{attribute 'qualified_only'}
VAR_GLOBAL
	calc0: LREAL :=  10;
	calc1: LREAL :=  10;
	calc2: LREAL :=  10;
	calc3: LREAL :=  10;
	calc4: LREAL :=  10;
	calc5: LREAL :=  10;
	calc6: LREAL :=  10;
	calc7: LREAL :=  10;
	calc8: LREAL :=  10;
	calc9: LREAL :=  10;
	calc10: LREAL :=  10;
	calc11: LREAL :=  10;
	calc12: LREAL :=  10;
	calc13: LREAL :=  10;
	calc14: LREAL :=  10;
	calc15: LREAL :=  10;
	calc16: LREAL :=  10;
	calc17: LREAL :=  10;
	calc18: LREAL :=  10;
	calc19: LREAL :=  10;
	calc20: LREAL :=  10;
	calc21: LREAL :=  10;
	calc22: LREAL :=  10;
	calc23: LREAL :=  10;
	calc24: LREAL :=  10;
	calc25: LREAL :=  10;
	calc26: LREAL :=  10;
	calc27: LREAL :=  10;
	calc28: LREAL :=  10;
	calc29: LREAL :=  10;
	calc30: LREAL :=  10;
	calc31: LREAL :=  10;
	calc32: LREAL :=  10;
	calc33: LREAL :=  10;
	calc34: LREAL :=  10;
	calc35: LREAL :=  10;
	calc36: LREAL :=  10;
	calc37: LREAL :=  10;
	calc38: LREAL :=  10;
	calc39: LREAL :=  10;
	calc40: LREAL :=  10;
	calc41: LREAL :=  10;
	calc42: LREAL :=  10;
	calc43: LREAL :=  10;
	calc44: LREAL :=  10;
	calc45: LREAL :=  10;
	calc46: LREAL :=  10;
	calc47: LREAL :=  10;
	calc48: LREAL :=  10;
	calc49: LREAL :=  10;
	calc50: LREAL :=  10;
	calc51: LREAL :=  10;
	calc52: LREAL :=  10;
	calc53: LREAL :=  10;
	calc54: LREAL :=  10;
	calc55: LREAL :=  10;
	calc56: LREAL :=  10;
	calc57: LREAL :=  10;
	calc58: LREAL :=  10;
	calc59: LREAL :=  10;
	calc60: LREAL :=  10;
	calc61: LREAL :=  10;
	calc62: LREAL :=  10;
	calc63: LREAL :=  10;
	calc64: LREAL :=  10;
	calc65: LREAL :=  10;
	calc66: LREAL :=  10;
	calc67: LREAL :=  10;
	calc68: LREAL :=  10;
	calc69: LREAL :=  10;
	calc70: LREAL :=  10;
	calc71: LREAL :=  10;
	calc72: LREAL :=  10;
	calc73: LREAL :=  10;
	calc74: LREAL :=  10;
	calc75: LREAL :=  10;
	calc76: LREAL :=  10;
	calc77: LREAL :=  10;
	calc78: LREAL :=  10;
	calc79: LREAL :=  10;
	calc80: LREAL :=  10;
	calc81: LREAL :=  10;
	calc82: LREAL :=  10;
	calc83: LREAL :=  10;
	calc84: LREAL :=  10;
	calc85: LREAL :=  10;
	calc86: LREAL :=  10;
	calc87: LREAL :=  10;
	calc88: LREAL :=  10;
	calc89: LREAL :=  10;
	calc90: LREAL :=  10;
	calc91: LREAL :=  10;
	calc92: LREAL :=  10;
	calc93: LREAL :=  10;
	calc94: LREAL :=  10;
	calc95: LREAL :=  10;
	calc96: LREAL :=  10;
	calc97: LREAL :=  10;
	calc98: LREAL :=  10;
	calc99: LREAL :=  10;
	calc100: LREAL :=  10;
	calc101: LREAL :=  10;
	calc102: LREAL :=  10;
	calc103: LREAL :=  10;
	calc104: LREAL :=  10;
	calc105: LREAL :=  10;
	calc106: LREAL :=  10;
	calc107: LREAL :=  10;
	calc108: LREAL :=  10;
	calc109: LREAL :=  10;
	calc110: LREAL :=  10;
	calc111: LREAL :=  10;
	calc112: LREAL :=  10;
	calc113: LREAL :=  10;
	calc114: LREAL :=  10;
	calc115: LREAL :=  10;
	calc116: LREAL :=  10;
	calc117: LREAL :=  10;
	calc118: LREAL :=  10;
	calc119: LREAL :=  10;
	calc120: LREAL :=  10;
	calc121: LREAL :=  10;
	calc122: LREAL :=  10;
	calc123: LREAL :=  10;
	calc124: LREAL :=  10;
	calc125: LREAL :=  10;
	calc126: LREAL :=  10;
	calc127: LREAL :=  10;
	calc128: LREAL :=  10;
	calc129: LREAL :=  10;
	calc130: LREAL :=  10;
	calc131: LREAL :=  10;
	calc132: LREAL :=  10;
	calc133: LREAL :=  10;
	calc134: LREAL :=  10;
	calc135: LREAL :=  10;
	calc136: LREAL :=  10;
	calc137: LREAL :=  10;
	calc138: LREAL :=  10;
	calc139: LREAL :=  10;
	calc140: LREAL :=  10;
	calc141: LREAL :=  10;
	calc142: LREAL :=  10;
	calc143: LREAL :=  10;
	calc144: LREAL :=  10;
	calc145: LREAL :=  10;
	calc146: LREAL :=  10;
	calc147: LREAL :=  10;
	calc148: LREAL :=  10;
	calc149: LREAL :=  10;
	calc150: LREAL :=  10;
	calc151: LREAL :=  10;
	calc152: LREAL :=  10;
	calc153: LREAL :=  10;
	calc154: LREAL :=  10;
	calc155: LREAL :=  10;
	calc156: LREAL :=  10;
	calc157: LREAL :=  10;
	calc158: LREAL :=  10;
	calc159: LREAL :=  10;
	calc160: LREAL :=  10;
	calc161: LREAL :=  10;
	calc162: LREAL :=  10;
	calc163: LREAL :=  10;
	calc164: LREAL :=  10;
	calc165: LREAL :=  10;
	calc166: LREAL :=  10;
	calc167: LREAL :=  10;
	calc168: LREAL :=  10;
	calc169: LREAL :=  10;
	calc170: LREAL :=  10;
	calc171: LREAL :=  10;
	calc172: LREAL :=  10;
	calc173: LREAL :=  10;
	calc174: LREAL :=  10;
	calc175: LREAL :=  10;
	calc176: LREAL :=  10;
	calc177: LREAL :=  10;
	calc178: LREAL :=  10;
	calc179: LREAL :=  10;
	calc180: LREAL :=  10;
	calc181: LREAL :=  10;
	calc182: LREAL :=  10;
	calc183: LREAL :=  10;
	calc184: LREAL :=  10;
	calc185: LREAL :=  10;
	calc186: LREAL :=  10;
	calc187: LREAL :=  10;
	calc188: LREAL :=  10;
	calc189: LREAL :=  10;
	calc190: LREAL :=  10;
	calc191: LREAL :=  10;
	calc192: LREAL :=  10;
	calc193: LREAL :=  10;
	calc194: LREAL :=  10;
	calc195: LREAL :=  10;
	calc196: LREAL :=  10;
	calc197: LREAL :=  10;
	calc198: LREAL :=  10;
	calc199: LREAL :=  10;
	calc200: LREAL :=  10;
	calc201: LREAL :=  10;
	calc202: LREAL :=  10;
	calc203: LREAL :=  10;
	calc204: LREAL :=  10;
	calc205: LREAL :=  10;
	calc206: LREAL :=  10;
	calc207: LREAL :=  10;
	calc208: LREAL :=  10;
	calc209: LREAL :=  10;
	calc210: LREAL :=  10;
	calc211: LREAL :=  10;
	calc212: LREAL :=  10;
	calc213: LREAL :=  10;
	calc214: LREAL :=  10;
	calc215: LREAL :=  10;
	calc216: LREAL :=  10;
	calc217: LREAL :=  10;
	calc218: LREAL :=  10;
	calc219: LREAL :=  10;
	calc220: LREAL :=  10;
	calc221: LREAL :=  10;
	calc222: LREAL :=  10;
	calc223: LREAL :=  10;
	calc224: LREAL :=  10;
	calc225: LREAL :=  10;
	calc226: LREAL :=  10;
	calc227: LREAL :=  10;
	calc228: LREAL :=  10;
	calc229: LREAL :=  10;
	calc230: LREAL :=  10;
	calc231: LREAL :=  10;
	calc232: LREAL :=  10;
	calc233: LREAL :=  10;
	calc234: LREAL :=  10;
	calc235: LREAL :=  10;
	calc236: LREAL :=  10;
	calc237: LREAL :=  10;
	calc238: LREAL :=  10;
	calc239: LREAL :=  10;
	calc240: LREAL :=  10;
	calc241: LREAL :=  10;
	calc242: LREAL :=  10;
	calc243: LREAL :=  10;
	calc244: LREAL :=  10;
	calc245: LREAL :=  10;
	calc246: LREAL :=  10;
	calc247: LREAL :=  10;
	calc248: LREAL :=  10;
	calc249: LREAL :=  10;
	calc250: LREAL :=  10;
	calc251: LREAL :=  10;
	calc252: LREAL :=  10;
	calc253: LREAL :=  10;
	calc254: LREAL :=  10;
	calc255: LREAL :=  10;
	calc256: LREAL :=  10;
	calc257: LREAL :=  10;
	calc258: LREAL :=  10;
	calc259: LREAL :=  10;
	calc260: LREAL :=  10;
	calc261: LREAL :=  10;
	calc262: LREAL :=  10;
	calc263: LREAL :=  10;
	calc264: LREAL :=  10;
	calc265: LREAL :=  10;
	calc266: LREAL :=  10;
	calc267: LREAL :=  10;
	calc268: LREAL :=  10;
	calc269: LREAL :=  10;
	calc270: LREAL :=  10;
	calc271: LREAL :=  10;
	calc272: LREAL :=  10;
	calc273: LREAL :=  10;
	calc274: LREAL :=  10;
	calc275: LREAL :=  10;
	calc276: LREAL :=  10;
	calc277: LREAL :=  10;
	calc278: LREAL :=  10;
	calc279: LREAL :=  10;
	calc280: LREAL :=  10;
	calc281: LREAL :=  10;
	calc282: LREAL :=  10;
	calc283: LREAL :=  10;
	calc284: LREAL :=  10;
	calc285: LREAL :=  10;
	calc286: LREAL :=  10;
	calc287: LREAL :=  10;
	calc288: LREAL :=  10;
	calc289: LREAL :=  10;
	calc290: LREAL :=  10;
	calc291: LREAL :=  10;
	calc292: LREAL :=  10;
	calc293: LREAL :=  10;
	calc294: LREAL :=  10;
	calc295: LREAL :=  10;
	calc296: LREAL :=  10;
	calc297: LREAL :=  10;
	calc298: LREAL :=  10;
	calc299: LREAL :=  10;
	calc300: LREAL :=  10;
	calc301: LREAL :=  10;
	calc302: LREAL :=  10;
	calc303: LREAL :=  10;
	calc304: LREAL :=  10;
	calc305: LREAL :=  10;
	calc306: LREAL :=  10;
	calc307: LREAL :=  10;
	calc308: LREAL :=  10;
	calc309: LREAL :=  10;
	calc310: LREAL :=  10;
	calc311: LREAL :=  10;
	calc312: LREAL :=  10;
	calc313: LREAL :=  10;
	calc314: LREAL :=  10;
	calc315: LREAL :=  10;
	calc316: LREAL :=  10;
	calc317: LREAL :=  10;
	calc318: LREAL :=  10;
	calc319: LREAL :=  10;
	calc320: LREAL :=  10;
	calc321: LREAL :=  10;
	calc322: LREAL :=  10;
	calc323: LREAL :=  10;
	calc324: LREAL :=  10;
	calc325: LREAL :=  10;
	calc326: LREAL :=  10;
	calc327: LREAL :=  10;
	calc328: LREAL :=  10;
	calc329: LREAL :=  10;
	calc330: LREAL :=  10;
	calc331: LREAL :=  10;
	calc332: LREAL :=  10;
	calc333: LREAL :=  10;
	calc334: LREAL :=  10;
	calc335: LREAL :=  10;
	calc336: LREAL :=  10;
	calc337: LREAL :=  10;
	calc338: LREAL :=  10;
	calc339: LREAL :=  10;
	calc340: LREAL :=  10;
	calc341: LREAL :=  10;
	calc342: LREAL :=  10;
	calc343: LREAL :=  10;
	calc344: LREAL :=  10;
	calc345: LREAL :=  10;
	calc346: LREAL :=  10;
	calc347: LREAL :=  10;
	calc348: LREAL :=  10;
	calc349: LREAL :=  10;
	calc350: LREAL :=  10;
	calc351: LREAL :=  10;
	calc352: LREAL :=  10;
	calc353: LREAL :=  10;
	calc354: LREAL :=  10;
	calc355: LREAL :=  10;
	calc356: LREAL :=  10;
	calc357: LREAL :=  10;
	calc358: LREAL :=  10;
	calc359: LREAL :=  10;
	calc360: LREAL :=  10;
	calc361: LREAL :=  10;
	calc362: LREAL :=  10;
	calc363: LREAL :=  10;
	calc364: LREAL :=  10;
	calc365: LREAL :=  10;
	calc366: LREAL :=  10;
	calc367: LREAL :=  10;
	calc368: LREAL :=  10;
	calc369: LREAL :=  10;
	calc370: LREAL :=  10;
	calc371: LREAL :=  10;
	calc372: LREAL :=  10;
	calc373: LREAL :=  10;
	calc374: LREAL :=  10;
	calc375: LREAL :=  10;
	calc376: LREAL :=  10;
	calc377: LREAL :=  10;
	calc378: LREAL :=  10;
	calc379: LREAL :=  10;
	calc380: LREAL :=  10;
	calc381: LREAL :=  10;
	calc382: LREAL :=  10;
	calc383: LREAL :=  10;
	calc384: LREAL :=  10;
	calc385: LREAL :=  10;
	calc386: LREAL :=  10;
	calc387: LREAL :=  10;
	calc388: LREAL :=  10;
	calc389: LREAL :=  10;
	calc390: LREAL :=  10;
	calc391: LREAL :=  10;
	calc392: LREAL :=  10;
	calc393: LREAL :=  10;
	calc394: LREAL :=  10;
	calc395: LREAL :=  10;
	calc396: LREAL :=  10;
	calc397: LREAL :=  10;
	calc398: LREAL :=  10;
	calc399: LREAL :=  10;
	calc400: LREAL :=  10;
	calc401: LREAL :=  10;
	calc402: LREAL :=  10;
	calc403: LREAL :=  10;
	calc404: LREAL :=  10;
	calc405: LREAL :=  10;
	calc406: LREAL :=  10;
	calc407: LREAL :=  10;
	calc408: LREAL :=  10;
	calc409: LREAL :=  10;
	calc410: LREAL :=  10;
	calc411: LREAL :=  10;
	calc412: LREAL :=  10;
	calc413: LREAL :=  10;
	calc414: LREAL :=  10;
	calc415: LREAL :=  10;
	calc416: LREAL :=  10;
	calc417: LREAL :=  10;
	calc418: LREAL :=  10;
	calc419: LREAL :=  10;
	calc420: LREAL :=  10;
	calc421: LREAL :=  10;
	calc422: LREAL :=  10;
	calc423: LREAL :=  10;
	calc424: LREAL :=  10;
	calc425: LREAL :=  10;
	calc426: LREAL :=  10;
	calc427: LREAL :=  10;
	calc428: LREAL :=  10;
	calc429: LREAL :=  10;
	calc430: LREAL :=  10;
	calc431: LREAL :=  10;
	calc432: LREAL :=  10;
	calc433: LREAL :=  10;
	calc434: LREAL :=  10;
	calc435: LREAL :=  10;
	calc436: LREAL :=  10;
	calc437: LREAL :=  10;
	calc438: LREAL :=  10;
	calc439: LREAL :=  10;
	calc440: LREAL :=  10;
	calc441: LREAL :=  10;
	calc442: LREAL :=  10;
	calc443: LREAL :=  10;
	calc444: LREAL :=  10;
	calc445: LREAL :=  10;
	calc446: LREAL :=  10;
	calc447: LREAL :=  10;
	calc448: LREAL :=  10;
	calc449: LREAL :=  10;
	calc450: LREAL :=  10;
	calc451: LREAL :=  10;
	calc452: LREAL :=  10;
	calc453: LREAL :=  10;
	calc454: LREAL :=  10;
	calc455: LREAL :=  10;
	calc456: LREAL :=  10;
	calc457: LREAL :=  10;
	calc458: LREAL :=  10;
	calc459: LREAL :=  10;
	calc460: LREAL :=  10;
	calc461: LREAL :=  10;
	calc462: LREAL :=  10;
	calc463: LREAL :=  10;
	calc464: LREAL :=  10;
	calc465: LREAL :=  10;
	calc466: LREAL :=  10;
	calc467: LREAL :=  10;
	calc468: LREAL :=  10;
	calc469: LREAL :=  10;
	calc470: LREAL :=  10;
	calc471: LREAL :=  10;
	calc472: LREAL :=  10;
	calc473: LREAL :=  10;
	calc474: LREAL :=  10;
	calc475: LREAL :=  10;
	calc476: LREAL :=  10;
	calc477: LREAL :=  10;
	calc478: LREAL :=  10;
	calc479: LREAL :=  10;
	calc480: LREAL :=  10;
	calc481: LREAL :=  10;
	calc482: LREAL :=  10;
	calc483: LREAL :=  10;
	calc484: LREAL :=  10;
	calc485: LREAL :=  10;
	calc486: LREAL :=  10;
	calc487: LREAL :=  10;
	calc488: LREAL :=  10;
	calc489: LREAL :=  10;
	calc490: LREAL :=  10;
	calc491: LREAL :=  10;
	calc492: LREAL :=  10;
	calc493: LREAL :=  10;
	calc494: LREAL :=  10;
	calc495: LREAL :=  10;
	calc496: LREAL :=  10;
	calc497: LREAL :=  10;
	calc498: LREAL :=  10;
	calc499: LREAL :=  10;
	calc500: LREAL :=  10;
	calc501: LREAL :=  10;
	calc502: LREAL :=  10;
	calc503: LREAL :=  10;
	calc504: LREAL :=  10;
	calc505: LREAL :=  10;
	calc506: LREAL :=  10;
	calc507: LREAL :=  10;
	calc508: LREAL :=  10;
	calc509: LREAL :=  10;
	calc510: LREAL :=  10;
	calc511: LREAL :=  10;
	calc512: LREAL :=  10;
	calc513: LREAL :=  10;
	calc514: LREAL :=  10;
	calc515: LREAL :=  10;
	calc516: LREAL :=  10;
	calc517: LREAL :=  10;
	calc518: LREAL :=  10;
	calc519: LREAL :=  10;
	calc520: LREAL :=  10;
	calc521: LREAL :=  10;
	calc522: LREAL :=  10;
	calc523: LREAL :=  10;
	calc524: LREAL :=  10;
	calc525: LREAL :=  10;
	calc526: LREAL :=  10;
	calc527: LREAL :=  10;
	calc528: LREAL :=  10;
	calc529: LREAL :=  10;
	calc530: LREAL :=  10;
	calc531: LREAL :=  10;
	calc532: LREAL :=  10;
	calc533: LREAL :=  10;
	calc534: LREAL :=  10;
	calc535: LREAL :=  10;
	calc536: LREAL :=  10;
	calc537: LREAL :=  10;
	calc538: LREAL :=  10;
	calc539: LREAL :=  10;
	calc540: LREAL :=  10;
	calc541: LREAL :=  10;
	calc542: LREAL :=  10;
	calc543: LREAL :=  10;
	calc544: LREAL :=  10;
	calc545: LREAL :=  10;
	calc546: LREAL :=  10;
	calc547: LREAL :=  10;
	calc548: LREAL :=  10;
	calc549: LREAL :=  10;
	calc550: LREAL :=  10;
	calc551: LREAL :=  10;
	calc552: LREAL :=  10;
	calc553: LREAL :=  10;
	calc554: LREAL :=  10;
	calc555: LREAL :=  10;
	calc556: LREAL :=  10;
	calc557: LREAL :=  10;
	calc558: LREAL :=  10;
	calc559: LREAL :=  10;
	calc560: LREAL :=  10;
	calc561: LREAL :=  10;
	calc562: LREAL :=  10;
	calc563: LREAL :=  10;
	calc564: LREAL :=  10;
	calc565: LREAL :=  10;
	calc566: LREAL :=  10;
	calc567: LREAL :=  10;
	calc568: LREAL :=  10;
	calc569: LREAL :=  10;
	calc570: LREAL :=  10;
	calc571: LREAL :=  10;
	calc572: LREAL :=  10;
	calc573: LREAL :=  10;
	calc574: LREAL :=  10;
	calc575: LREAL :=  10;
	calc576: LREAL :=  10;
	calc577: LREAL :=  10;
	calc578: LREAL :=  10;
	calc579: LREAL :=  10;
	calc580: LREAL :=  10;
	calc581: LREAL :=  10;
	calc582: LREAL :=  10;
	calc583: LREAL :=  10;
	calc584: LREAL :=  10;
	calc585: LREAL :=  10;
	calc586: LREAL :=  10;
	calc587: LREAL :=  10;
	calc588: LREAL :=  10;
	calc589: LREAL :=  10;
	calc590: LREAL :=  10;
	calc591: LREAL :=  10;
	calc592: LREAL :=  10;
	calc593: LREAL :=  10;
	calc594: LREAL :=  10;
	calc595: LREAL :=  10;
	calc596: LREAL :=  10;
	calc597: LREAL :=  10;
	calc598: LREAL :=  10;
	calc599: LREAL :=  10;
	calc600: LREAL :=  10;
	calc601: LREAL :=  10;
	calc602: LREAL :=  10;
	calc603: LREAL :=  10;
	calc604: LREAL :=  10;
	calc605: LREAL :=  10;
	calc606: LREAL :=  10;
	calc607: LREAL :=  10;
	calc608: LREAL :=  10;
	calc609: LREAL :=  10;
	calc610: LREAL :=  10;
	calc611: LREAL :=  10;
	calc612: LREAL :=  10;
	calc613: LREAL :=  10;
	calc614: LREAL :=  10;
	calc615: LREAL :=  10;
	calc616: LREAL :=  10;
	calc617: LREAL :=  10;
	calc618: LREAL :=  10;
	calc619: LREAL :=  10;
	calc620: LREAL :=  10;
	calc621: LREAL :=  10;
	calc622: LREAL :=  10;
	calc623: LREAL :=  10;
	calc624: LREAL :=  10;
	calc625: LREAL :=  10;
	calc626: LREAL :=  10;
	calc627: LREAL :=  10;
	calc628: LREAL :=  10;
	calc629: LREAL :=  10;
	calc630: LREAL :=  10;
	calc631: LREAL :=  10;
	calc632: LREAL :=  10;
	calc633: LREAL :=  10;
	calc634: LREAL :=  10;
	calc635: LREAL :=  10;
	calc636: LREAL :=  10;
	calc637: LREAL :=  10;
	calc638: LREAL :=  10;
	calc639: LREAL :=  10;
	calc640: LREAL :=  10;
	calc641: LREAL :=  10;
	calc642: LREAL :=  10;
	calc643: LREAL :=  10;
	calc644: LREAL :=  10;
	calc645: LREAL :=  10;
	calc646: LREAL :=  10;
	calc647: LREAL :=  10;
	calc648: LREAL :=  10;
	calc649: LREAL :=  10;
	calc650: LREAL :=  10;
	calc651: LREAL :=  10;
	calc652: LREAL :=  10;
	calc653: LREAL :=  10;
	calc654: LREAL :=  10;
	calc655: LREAL :=  10;
	calc656: LREAL :=  10;
	calc657: LREAL :=  10;
	calc658: LREAL :=  10;
	calc659: LREAL :=  10;
	calc660: LREAL :=  10;
	calc661: LREAL :=  10;
	calc662: LREAL :=  10;
	calc663: LREAL :=  10;
	calc664: LREAL :=  10;
	calc665: LREAL :=  10;
	calc666: LREAL :=  10;
	calc667: LREAL :=  10;
	calc668: LREAL :=  10;
	calc669: LREAL :=  10;
	calc670: LREAL :=  10;
	calc671: LREAL :=  10;
	calc672: LREAL :=  10;
	calc673: LREAL :=  10;
	calc674: LREAL :=  10;
	calc675: LREAL :=  10;
	calc676: LREAL :=  10;
	calc677: LREAL :=  10;
	calc678: LREAL :=  10;
	calc679: LREAL :=  10;
	calc680: LREAL :=  10;
	calc681: LREAL :=  10;
	calc682: LREAL :=  10;
	calc683: LREAL :=  10;
	calc684: LREAL :=  10;
	calc685: LREAL :=  10;
	calc686: LREAL :=  10;
	calc687: LREAL :=  10;
	calc688: LREAL :=  10;
	calc689: LREAL :=  10;
	calc690: LREAL :=  10;
	calc691: LREAL :=  10;
	calc692: LREAL :=  10;
	calc693: LREAL :=  10;
	calc694: LREAL :=  10;
	calc695: LREAL :=  10;
	calc696: LREAL :=  10;
	calc697: LREAL :=  10;
	calc698: LREAL :=  10;
	calc699: LREAL :=  10;
	calc700: LREAL :=  10;
	calc701: LREAL :=  10;
	calc702: LREAL :=  10;
	calc703: LREAL :=  10;
	calc704: LREAL :=  10;
	calc705: LREAL :=  10;
	calc706: LREAL :=  10;
	calc707: LREAL :=  10;
	calc708: LREAL :=  10;
	calc709: LREAL :=  10;
	calc710: LREAL :=  10;
	calc711: LREAL :=  10;
	calc712: LREAL :=  10;
	calc713: LREAL :=  10;
	calc714: LREAL :=  10;
	calc715: LREAL :=  10;
	calc716: LREAL :=  10;
	calc717: LREAL :=  10;
	calc718: LREAL :=  10;
	calc719: LREAL :=  10;
	calc720: LREAL :=  10;
	calc721: LREAL :=  10;
	calc722: LREAL :=  10;
	calc723: LREAL :=  10;
	calc724: LREAL :=  10;
	calc725: LREAL :=  10;
	calc726: LREAL :=  10;
	calc727: LREAL :=  10;
	calc728: LREAL :=  10;
	calc729: LREAL :=  10;
	calc730: LREAL :=  10;
	calc731: LREAL :=  10;
	calc732: LREAL :=  10;
	calc733: LREAL :=  10;
	calc734: LREAL :=  10;
	calc735: LREAL :=  10;
	calc736: LREAL :=  10;
	calc737: LREAL :=  10;
	calc738: LREAL :=  10;
	calc739: LREAL :=  10;
	calc740: LREAL :=  10;
	calc741: LREAL :=  10;
	calc742: LREAL :=  10;
	calc743: LREAL :=  10;
	calc744: LREAL :=  10;
	calc745: LREAL :=  10;
	calc746: LREAL :=  10;
	calc747: LREAL :=  10;
	calc748: LREAL :=  10;
	calc749: LREAL :=  10;
	calc750: LREAL :=  10;
	calc751: LREAL :=  10;
	calc752: LREAL :=  10;
	calc753: LREAL :=  10;
	calc754: LREAL :=  10;
	calc755: LREAL :=  10;
	calc756: LREAL :=  10;
	calc757: LREAL :=  10;
	calc758: LREAL :=  10;
	calc759: LREAL :=  10;
	calc760: LREAL :=  10;
	calc761: LREAL :=  10;
	calc762: LREAL :=  10;
	calc763: LREAL :=  10;
	calc764: LREAL :=  10;
	calc765: LREAL :=  10;
	calc766: LREAL :=  10;
	calc767: LREAL :=  10;
	calc768: LREAL :=  10;
	calc769: LREAL :=  10;
	calc770: LREAL :=  10;
	calc771: LREAL :=  10;
	calc772: LREAL :=  10;
	calc773: LREAL :=  10;
	calc774: LREAL :=  10;
	calc775: LREAL :=  10;
	calc776: LREAL :=  10;
	calc777: LREAL :=  10;
	calc778: LREAL :=  10;
	calc779: LREAL :=  10;
	calc780: LREAL :=  10;
	calc781: LREAL :=  10;
	calc782: LREAL :=  10;
	calc783: LREAL :=  10;
	calc784: LREAL :=  10;
	calc785: LREAL :=  10;
	calc786: LREAL :=  10;
	calc787: LREAL :=  10;
	calc788: LREAL :=  10;
	calc789: LREAL :=  10;
	calc790: LREAL :=  10;
	calc791: LREAL :=  10;
	calc792: LREAL :=  10;
	calc793: LREAL :=  10;
	calc794: LREAL :=  10;
	calc795: LREAL :=  10;
	calc796: LREAL :=  10;
	calc797: LREAL :=  10;
	calc798: LREAL :=  10;
	calc799: LREAL :=  10;
	calc800: LREAL :=  10;
	calc801: LREAL :=  10;
	calc802: LREAL :=  10;
	calc803: LREAL :=  10;
	calc804: LREAL :=  10;
	calc805: LREAL :=  10;
	calc806: LREAL :=  10;
	calc807: LREAL :=  10;
	calc808: LREAL :=  10;
	calc809: LREAL :=  10;
	calc810: LREAL :=  10;
	calc811: LREAL :=  10;
	calc812: LREAL :=  10;
	calc813: LREAL :=  10;
	calc814: LREAL :=  10;
	calc815: LREAL :=  10;
	calc816: LREAL :=  10;
	calc817: LREAL :=  10;
	calc818: LREAL :=  10;
	calc819: LREAL :=  10;
	calc820: LREAL :=  10;
	calc821: LREAL :=  10;
	calc822: LREAL :=  10;
	calc823: LREAL :=  10;
	calc824: LREAL :=  10;
	calc825: LREAL :=  10;
	calc826: LREAL :=  10;
	calc827: LREAL :=  10;
	calc828: LREAL :=  10;
	calc829: LREAL :=  10;
	calc830: LREAL :=  10;
	calc831: LREAL :=  10;
	calc832: LREAL :=  10;
	calc833: LREAL :=  10;
	calc834: LREAL :=  10;
	calc835: LREAL :=  10;
	calc836: LREAL :=  10;
	calc837: LREAL :=  10;
	calc838: LREAL :=  10;
	calc839: LREAL :=  10;
	calc840: LREAL :=  10;
	calc841: LREAL :=  10;
	calc842: LREAL :=  10;
	calc843: LREAL :=  10;
	calc844: LREAL :=  10;
	calc845: LREAL :=  10;
	calc846: LREAL :=  10;
	calc847: LREAL :=  10;
	calc848: LREAL :=  10;
	calc849: LREAL :=  10;
	calc850: LREAL :=  10;
	calc851: LREAL :=  10;
	calc852: LREAL :=  10;
	calc853: LREAL :=  10;
	calc854: LREAL :=  10;
	calc855: LREAL :=  10;
	calc856: LREAL :=  10;
	calc857: LREAL :=  10;
	calc858: LREAL :=  10;
	calc859: LREAL :=  10;
	calc860: LREAL :=  10;
	calc861: LREAL :=  10;
	calc862: LREAL :=  10;
	calc863: LREAL :=  10;
	calc864: LREAL :=  10;
	calc865: LREAL :=  10;
	calc866: LREAL :=  10;
	calc867: LREAL :=  10;
	calc868: LREAL :=  10;
	calc869: LREAL :=  10;
	calc870: LREAL :=  10;
	calc871: LREAL :=  10;
	calc872: LREAL :=  10;
	calc873: LREAL :=  10;
	calc874: LREAL :=  10;
	calc875: LREAL :=  10;
	calc876: LREAL :=  10;
	calc877: LREAL :=  10;
	calc878: LREAL :=  10;
	calc879: LREAL :=  10;
	calc880: LREAL :=  10;
	calc881: LREAL :=  10;
	calc882: LREAL :=  10;
	calc883: LREAL :=  10;
	calc884: LREAL :=  10;
	calc885: LREAL :=  10;
	calc886: LREAL :=  10;
	calc887: LREAL :=  10;
	calc888: LREAL :=  10;
	calc889: LREAL :=  10;
	calc890: LREAL :=  10;
	calc891: LREAL :=  10;
	calc892: LREAL :=  10;
	calc893: LREAL :=  10;
	calc894: LREAL :=  10;
	calc895: LREAL :=  10;
	calc896: LREAL :=  10;
	calc897: LREAL :=  10;
	calc898: LREAL :=  10;
	calc899: LREAL :=  10;
	calc900: LREAL :=  10;
	calc901: LREAL :=  10;
	calc902: LREAL :=  10;
	calc903: LREAL :=  10;
	calc904: LREAL :=  10;
	calc905: LREAL :=  10;
	calc906: LREAL :=  10;
	calc907: LREAL :=  10;
	calc908: LREAL :=  10;
	calc909: LREAL :=  10;
	calc910: LREAL :=  10;
	calc911: LREAL :=  10;
	calc912: LREAL :=  10;
	calc913: LREAL :=  10;
	calc914: LREAL :=  10;
	calc915: LREAL :=  10;
	calc916: LREAL :=  10;
	calc917: LREAL :=  10;
	calc918: LREAL :=  10;
	calc919: LREAL :=  10;
	calc920: LREAL :=  10;
	calc921: LREAL :=  10;
	calc922: LREAL :=  10;
	calc923: LREAL :=  10;
	calc924: LREAL :=  10;
	calc925: LREAL :=  10;
	calc926: LREAL :=  10;
	calc927: LREAL :=  10;
	calc928: LREAL :=  10;
	calc929: LREAL :=  10;
	calc930: LREAL :=  10;
	calc931: LREAL :=  10;
	calc932: LREAL :=  10;
	calc933: LREAL :=  10;
	calc934: LREAL :=  10;
	calc935: LREAL :=  10;
	calc936: LREAL :=  10;
	calc937: LREAL :=  10;
	calc938: LREAL :=  10;
	calc939: LREAL :=  10;
	calc940: LREAL :=  10;
	calc941: LREAL :=  10;
	calc942: LREAL :=  10;
	calc943: LREAL :=  10;
	calc944: LREAL :=  10;
	calc945: LREAL :=  10;
	calc946: LREAL :=  10;
	calc947: LREAL :=  10;
	calc948: LREAL :=  10;
	calc949: LREAL :=  10;
	calc950: LREAL :=  10;
	calc951: LREAL :=  10;
	calc952: LREAL :=  10;
	calc953: LREAL :=  10;
	calc954: LREAL :=  10;
	calc955: LREAL :=  10;
	calc956: LREAL :=  10;
	calc957: LREAL :=  10;
	calc958: LREAL :=  10;
	calc959: LREAL :=  10;
	calc960: LREAL :=  10;
	calc961: LREAL :=  10;
	calc962: LREAL :=  10;
	calc963: LREAL :=  10;
	calc964: LREAL :=  10;
	calc965: LREAL :=  10;
	calc966: LREAL :=  10;
	calc967: LREAL :=  10;
	calc968: LREAL :=  10;
	calc969: LREAL :=  10;
	calc970: LREAL :=  10;
	calc971: LREAL :=  10;
	calc972: LREAL :=  10;
	calc973: LREAL :=  10;
	calc974: LREAL :=  10;
	calc975: LREAL :=  10;
	calc976: LREAL :=  10;
	calc977: LREAL :=  10;
	calc978: LREAL :=  10;
	calc979: LREAL :=  10;
	calc980: LREAL :=  10;
	calc981: LREAL :=  10;
	calc982: LREAL :=  10;
	calc983: LREAL :=  10;
	calc984: LREAL :=  10;
	calc985: LREAL :=  10;
	calc986: LREAL :=  10;
	calc987: LREAL :=  10;
	calc988: LREAL :=  10;
	calc989: LREAL :=  10;
	calc990: LREAL :=  10;
	calc991: LREAL :=  10;
	calc992: LREAL :=  10;
	calc993: LREAL :=  10;
	calc994: LREAL :=  10;
	calc995: LREAL :=  10;
	calc996: LREAL :=  10;
	calc997: LREAL :=  10;
	calc998: LREAL :=  10;
	calc999: LREAL :=  10;
	calc1000: LREAL :=  10;
	calc1001: LREAL :=  10;
	calc1002: LREAL :=  10;
	calc1003: LREAL :=  10;
	calc1004: LREAL :=  10;
	calc1005: LREAL :=  10;
	calc1006: LREAL :=  10;
	calc1007: LREAL :=  10;
	calc1008: LREAL :=  10;
	calc1009: LREAL :=  10;
	calc1010: LREAL :=  10;
	calc1011: LREAL :=  10;
	calc1012: LREAL :=  10;
	calc1013: LREAL :=  10;
	calc1014: LREAL :=  10;
	calc1015: LREAL :=  10;
	calc1016: LREAL :=  10;
	calc1017: LREAL :=  10;
	calc1018: LREAL :=  10;
	calc1019: LREAL :=  10;
	calc1020: LREAL :=  10;
	calc1021: LREAL :=  10;
	calc1022: LREAL :=  10;
	calc1023: LREAL :=  10;
	calc1024: LREAL :=  10;
	calc1025: LREAL :=  10;
	calc1026: LREAL :=  10;
	calc1027: LREAL :=  10;
	calc1028: LREAL :=  10;
	calc1029: LREAL :=  10;
	calc1030: LREAL :=  10;
	calc1031: LREAL :=  10;
	calc1032: LREAL :=  10;
	calc1033: LREAL :=  10;
	calc1034: LREAL :=  10;
	calc1035: LREAL :=  10;
	calc1036: LREAL :=  10;
	calc1037: LREAL :=  10;
	calc1038: LREAL :=  10;
	calc1039: LREAL :=  10;
	calc1040: LREAL :=  10;
	calc1041: LREAL :=  10;
	calc1042: LREAL :=  10;
	calc1043: LREAL :=  10;
	calc1044: LREAL :=  10;
	calc1045: LREAL :=  10;
	calc1046: LREAL :=  10;
	calc1047: LREAL :=  10;
	calc1048: LREAL :=  10;
	calc1049: LREAL :=  10;
	calc1050: LREAL :=  10;
	calc1051: LREAL :=  10;
	calc1052: LREAL :=  10;
	calc1053: LREAL :=  10;
	calc1054: LREAL :=  10;
	calc1055: LREAL :=  10;
	calc1056: LREAL :=  10;
	calc1057: LREAL :=  10;
	calc1058: LREAL :=  10;
	calc1059: LREAL :=  10;
	calc1060: LREAL :=  10;
	calc1061: LREAL :=  10;
	calc1062: LREAL :=  10;
	calc1063: LREAL :=  10;
	calc1064: LREAL :=  10;
	calc1065: LREAL :=  10;
	calc1066: LREAL :=  10;
	calc1067: LREAL :=  10;
	calc1068: LREAL :=  10;
	calc1069: LREAL :=  10;
	calc1070: LREAL :=  10;
	calc1071: LREAL :=  10;
	calc1072: LREAL :=  10;
	calc1073: LREAL :=  10;
	calc1074: LREAL :=  10;
	calc1075: LREAL :=  10;
	calc1076: LREAL :=  10;
	calc1077: LREAL :=  10;
	calc1078: LREAL :=  10;
	calc1079: LREAL :=  10;
	calc1080: LREAL :=  10;
	calc1081: LREAL :=  10;
	calc1082: LREAL :=  10;
	calc1083: LREAL :=  10;
	calc1084: LREAL :=  10;
	calc1085: LREAL :=  10;
	calc1086: LREAL :=  10;
	calc1087: LREAL :=  10;
	calc1088: LREAL :=  10;
	calc1089: LREAL :=  10;
	calc1090: LREAL :=  10;
	calc1091: LREAL :=  10;
	calc1092: LREAL :=  10;
	calc1093: LREAL :=  10;
	calc1094: LREAL :=  10;
	calc1095: LREAL :=  10;
	calc1096: LREAL :=  10;
	calc1097: LREAL :=  10;
	calc1098: LREAL :=  10;
	calc1099: LREAL :=  10;
	calc1100: LREAL :=  10;
	calc1101: LREAL :=  10;
	calc1102: LREAL :=  10;
	calc1103: LREAL :=  10;
	calc1104: LREAL :=  10;
	calc1105: LREAL :=  10;
	calc1106: LREAL :=  10;
	calc1107: LREAL :=  10;
	calc1108: LREAL :=  10;
	calc1109: LREAL :=  10;
	calc1110: LREAL :=  10;
	calc1111: LREAL :=  10;
	calc1112: LREAL :=  10;
	calc1113: LREAL :=  10;
	calc1114: LREAL :=  10;
	calc1115: LREAL :=  10;
	calc1116: LREAL :=  10;
	calc1117: LREAL :=  10;
	calc1118: LREAL :=  10;
	calc1119: LREAL :=  10;
	calc1120: LREAL :=  10;
	calc1121: LREAL :=  10;
	calc1122: LREAL :=  10;
	calc1123: LREAL :=  10;
	calc1124: LREAL :=  10;
	calc1125: LREAL :=  10;
	calc1126: LREAL :=  10;
	calc1127: LREAL :=  10;
	calc1128: LREAL :=  10;
	calc1129: LREAL :=  10;
	calc1130: LREAL :=  10;
	calc1131: LREAL :=  10;
	calc1132: LREAL :=  10;
	calc1133: LREAL :=  10;
	calc1134: LREAL :=  10;
	calc1135: LREAL :=  10;
	calc1136: LREAL :=  10;
	calc1137: LREAL :=  10;
	calc1138: LREAL :=  10;
	calc1139: LREAL :=  10;
	calc1140: LREAL :=  10;
	calc1141: LREAL :=  10;
	calc1142: LREAL :=  10;
	calc1143: LREAL :=  10;
	calc1144: LREAL :=  10;
	calc1145: LREAL :=  10;
	calc1146: LREAL :=  10;
	calc1147: LREAL :=  10;
	calc1148: LREAL :=  10;
	calc1149: LREAL :=  10;
	calc1150: LREAL :=  10;
	calc1151: LREAL :=  10;
	calc1152: LREAL :=  10;
	calc1153: LREAL :=  10;
	calc1154: LREAL :=  10;
	calc1155: LREAL :=  10;
	calc1156: LREAL :=  10;
	calc1157: LREAL :=  10;
	calc1158: LREAL :=  10;
	calc1159: LREAL :=  10;
	calc1160: LREAL :=  10;
	calc1161: LREAL :=  10;
	calc1162: LREAL :=  10;
	calc1163: LREAL :=  10;
	calc1164: LREAL :=  10;
	calc1165: LREAL :=  10;
	calc1166: LREAL :=  10;
	calc1167: LREAL :=  10;
	calc1168: LREAL :=  10;
	calc1169: LREAL :=  10;
	calc1170: LREAL :=  10;
	calc1171: LREAL :=  10;
	calc1172: LREAL :=  10;
	calc1173: LREAL :=  10;
	calc1174: LREAL :=  10;
	calc1175: LREAL :=  10;
	calc1176: LREAL :=  10;
	calc1177: LREAL :=  10;
	calc1178: LREAL :=  10;
	calc1179: LREAL :=  10;
	calc1180: LREAL :=  10;
	calc1181: LREAL :=  10;
	calc1182: LREAL :=  10;
	calc1183: LREAL :=  10;
	calc1184: LREAL :=  10;
	calc1185: LREAL :=  10;
	calc1186: LREAL :=  10;
	calc1187: LREAL :=  10;
	calc1188: LREAL :=  10;
	calc1189: LREAL :=  10;
	calc1190: LREAL :=  10;
	calc1191: LREAL :=  10;
	calc1192: LREAL :=  10;
	calc1193: LREAL :=  10;
	calc1194: LREAL :=  10;
	calc1195: LREAL :=  10;
	calc1196: LREAL :=  10;
	calc1197: LREAL :=  10;
	calc1198: LREAL :=  10;
	calc1199: LREAL :=  10;
	calc1200: LREAL :=  10;
	calc1201: LREAL :=  10;
	calc1202: LREAL :=  10;
	calc1203: LREAL :=  10;
	calc1204: LREAL :=  10;
	calc1205: LREAL :=  10;
	calc1206: LREAL :=  10;
	calc1207: LREAL :=  10;
	calc1208: LREAL :=  10;
	calc1209: LREAL :=  10;
	calc1210: LREAL :=  10;
	calc1211: LREAL :=  10;
	calc1212: LREAL :=  10;
	calc1213: LREAL :=  10;
	calc1214: LREAL :=  10;
	calc1215: LREAL :=  10;
	calc1216: LREAL :=  10;
	calc1217: LREAL :=  10;
	calc1218: LREAL :=  10;
	calc1219: LREAL :=  10;
	calc1220: LREAL :=  10;
	calc1221: LREAL :=  10;
	calc1222: LREAL :=  10;
	calc1223: LREAL :=  10;
	calc1224: LREAL :=  10;
	calc1225: LREAL :=  10;
	calc1226: LREAL :=  10;
	calc1227: LREAL :=  10;
	calc1228: LREAL :=  10;
	calc1229: LREAL :=  10;
	calc1230: LREAL :=  10;
	calc1231: LREAL :=  10;
	calc1232: LREAL :=  10;
	calc1233: LREAL :=  10;
	calc1234: LREAL :=  10;
	calc1235: LREAL :=  10;
	calc1236: LREAL :=  10;
	calc1237: LREAL :=  10;
	calc1238: LREAL :=  10;
	calc1239: LREAL :=  10;
	calc1240: LREAL :=  10;
	calc1241: LREAL :=  10;
	calc1242: LREAL :=  10;
	calc1243: LREAL :=  10;
	calc1244: LREAL :=  10;
	calc1245: LREAL :=  10;
	calc1246: LREAL :=  10;
	calc1247: LREAL :=  10;
	calc1248: LREAL :=  10;
	calc1249: LREAL :=  10;
	calc1250: LREAL :=  10;
	calc1251: LREAL :=  10;
	calc1252: LREAL :=  10;
	calc1253: LREAL :=  10;
	calc1254: LREAL :=  10;
	calc1255: LREAL :=  10;
	calc1256: LREAL :=  10;
	calc1257: LREAL :=  10;
	calc1258: LREAL :=  10;
	calc1259: LREAL :=  10;
	calc1260: LREAL :=  10;
	calc1261: LREAL :=  10;
	calc1262: LREAL :=  10;
	calc1263: LREAL :=  10;
	calc1264: LREAL :=  10;
	calc1265: LREAL :=  10;
	calc1266: LREAL :=  10;
	calc1267: LREAL :=  10;
	calc1268: LREAL :=  10;
	calc1269: LREAL :=  10;
	calc1270: LREAL :=  10;
	calc1271: LREAL :=  10;
	calc1272: LREAL :=  10;
	calc1273: LREAL :=  10;
	calc1274: LREAL :=  10;
	calc1275: LREAL :=  10;
	calc1276: LREAL :=  10;
	calc1277: LREAL :=  10;
	calc1278: LREAL :=  10;
	calc1279: LREAL :=  10;
	calc1280: LREAL :=  10;
	calc1281: LREAL :=  10;
	calc1282: LREAL :=  10;
	calc1283: LREAL :=  10;
	calc1284: LREAL :=  10;
	calc1285: LREAL :=  10;
	calc1286: LREAL :=  10;
	calc1287: LREAL :=  10;
	calc1288: LREAL :=  10;
	calc1289: LREAL :=  10;
	calc1290: LREAL :=  10;
	calc1291: LREAL :=  10;
	calc1292: LREAL :=  10;
	calc1293: LREAL :=  10;
	calc1294: LREAL :=  10;
	calc1295: LREAL :=  10;
	calc1296: LREAL :=  10;
	calc1297: LREAL :=  10;
	calc1298: LREAL :=  10;
	calc1299: LREAL :=  10;
	calc1300: LREAL :=  10;
	calc1301: LREAL :=  10;
	calc1302: LREAL :=  10;
	calc1303: LREAL :=  10;
	calc1304: LREAL :=  10;
	calc1305: LREAL :=  10;
	calc1306: LREAL :=  10;
	calc1307: LREAL :=  10;
	calc1308: LREAL :=  10;
	calc1309: LREAL :=  10;
	calc1310: LREAL :=  10;
	calc1311: LREAL :=  10;
	calc1312: LREAL :=  10;
	calc1313: LREAL :=  10;
	calc1314: LREAL :=  10;
	calc1315: LREAL :=  10;
	calc1316: LREAL :=  10;
	calc1317: LREAL :=  10;
	calc1318: LREAL :=  10;
	calc1319: LREAL :=  10;
	calc1320: LREAL :=  10;
	calc1321: LREAL :=  10;
	calc1322: LREAL :=  10;
	calc1323: LREAL :=  10;
	calc1324: LREAL :=  10;
	calc1325: LREAL :=  10;
	calc1326: LREAL :=  10;
	calc1327: LREAL :=  10;
	calc1328: LREAL :=  10;
	calc1329: LREAL :=  10;
	calc1330: LREAL :=  10;
	calc1331: LREAL :=  10;
	calc1332: LREAL :=  10;
	calc1333: LREAL :=  10;
	calc1334: LREAL :=  10;
	calc1335: LREAL :=  10;
	calc1336: LREAL :=  10;
	calc1337: LREAL :=  10;
	calc1338: LREAL :=  10;
	calc1339: LREAL :=  10;
	calc1340: LREAL :=  10;
	calc1341: LREAL :=  10;
	calc1342: LREAL :=  10;
	calc1343: LREAL :=  10;
	calc1344: LREAL :=  10;
	calc1345: LREAL :=  10;
	calc1346: LREAL :=  10;
	calc1347: LREAL :=  10;
	calc1348: LREAL :=  10;
	calc1349: LREAL :=  10;
	calc1350: LREAL :=  10;
	calc1351: LREAL :=  10;
	calc1352: LREAL :=  10;
	calc1353: LREAL :=  10;
	calc1354: LREAL :=  10;
	calc1355: LREAL :=  10;
	calc1356: LREAL :=  10;
	calc1357: LREAL :=  10;
	calc1358: LREAL :=  10;
	calc1359: LREAL :=  10;
	calc1360: LREAL :=  10;
	calc1361: LREAL :=  10;
	calc1362: LREAL :=  10;
	calc1363: LREAL :=  10;
	calc1364: LREAL :=  10;
	calc1365: LREAL :=  10;
	calc1366: LREAL :=  10;
	calc1367: LREAL :=  10;
	calc1368: LREAL :=  10;
	calc1369: LREAL :=  10;
	calc1370: LREAL :=  10;
	calc1371: LREAL :=  10;
	calc1372: LREAL :=  10;
	calc1373: LREAL :=  10;
	calc1374: LREAL :=  10;
	calc1375: LREAL :=  10;
	calc1376: LREAL :=  10;
	calc1377: LREAL :=  10;
	calc1378: LREAL :=  10;
	calc1379: LREAL :=  10;
	calc1380: LREAL :=  10;
	calc1381: LREAL :=  10;
	calc1382: LREAL :=  10;
	calc1383: LREAL :=  10;
	calc1384: LREAL :=  10;
	calc1385: LREAL :=  10;
	calc1386: LREAL :=  10;
	calc1387: LREAL :=  10;
	calc1388: LREAL :=  10;
	calc1389: LREAL :=  10;
	calc1390: LREAL :=  10;
	calc1391: LREAL :=  10;
	calc1392: LREAL :=  10;
	calc1393: LREAL :=  10;
	calc1394: LREAL :=  10;
	calc1395: LREAL :=  10;
	calc1396: LREAL :=  10;
	calc1397: LREAL :=  10;
	calc1398: LREAL :=  10;
	calc1399: LREAL :=  10;
	calc1400: LREAL :=  10;
	calc1401: LREAL :=  10;
	calc1402: LREAL :=  10;
	calc1403: LREAL :=  10;
	calc1404: LREAL :=  10;
	calc1405: LREAL :=  10;
	calc1406: LREAL :=  10;
	calc1407: LREAL :=  10;
	calc1408: LREAL :=  10;
	calc1409: LREAL :=  10;
	calc1410: LREAL :=  10;
	calc1411: LREAL :=  10;
	calc1412: LREAL :=  10;
	calc1413: LREAL :=  10;
	calc1414: LREAL :=  10;
	calc1415: LREAL :=  10;
	calc1416: LREAL :=  10;
	calc1417: LREAL :=  10;
	calc1418: LREAL :=  10;
	calc1419: LREAL :=  10;
	calc1420: LREAL :=  10;
	calc1421: LREAL :=  10;
	calc1422: LREAL :=  10;
	calc1423: LREAL :=  10;
	calc1424: LREAL :=  10;
	calc1425: LREAL :=  10;
	calc1426: LREAL :=  10;
	calc1427: LREAL :=  10;
	calc1428: LREAL :=  10;
	calc1429: LREAL :=  10;
	calc1430: LREAL :=  10;
	calc1431: LREAL :=  10;
	calc1432: LREAL :=  10;
	calc1433: LREAL :=  10;
	calc1434: LREAL :=  10;
	calc1435: LREAL :=  10;
	calc1436: LREAL :=  10;
	calc1437: LREAL :=  10;
	calc1438: LREAL :=  10;
	calc1439: LREAL :=  10;
	calc1440: LREAL :=  10;
	calc1441: LREAL :=  10;
	calc1442: LREAL :=  10;
	calc1443: LREAL :=  10;
	calc1444: LREAL :=  10;
	calc1445: LREAL :=  10;
	calc1446: LREAL :=  10;
	calc1447: LREAL :=  10;
	calc1448: LREAL :=  10;
	calc1449: LREAL :=  10;
	calc1450: LREAL :=  10;
	calc1451: LREAL :=  10;
	calc1452: LREAL :=  10;
	calc1453: LREAL :=  10;
	calc1454: LREAL :=  10;
	calc1455: LREAL :=  10;
	calc1456: LREAL :=  10;
	calc1457: LREAL :=  10;
	calc1458: LREAL :=  10;
	calc1459: LREAL :=  10;
	calc1460: LREAL :=  10;
	calc1461: LREAL :=  10;
	calc1462: LREAL :=  10;
	calc1463: LREAL :=  10;
	calc1464: LREAL :=  10;
	calc1465: LREAL :=  10;
	calc1466: LREAL :=  10;
	calc1467: LREAL :=  10;
	calc1468: LREAL :=  10;
	calc1469: LREAL :=  10;
	calc1470: LREAL :=  10;
	calc1471: LREAL :=  10;
	calc1472: LREAL :=  10;
	calc1473: LREAL :=  10;
	calc1474: LREAL :=  10;
	calc1475: LREAL :=  10;
	calc1476: LREAL :=  10;
	calc1477: LREAL :=  10;
	calc1478: LREAL :=  10;
	calc1479: LREAL :=  10;
	calc1480: LREAL :=  10;
	calc1481: LREAL :=  10;
	calc1482: LREAL :=  10;
	calc1483: LREAL :=  10;
	calc1484: LREAL :=  10;
	calc1485: LREAL :=  10;
	calc1486: LREAL :=  10;
	calc1487: LREAL :=  10;
	calc1488: LREAL :=  10;
	calc1489: LREAL :=  10;
	calc1490: LREAL :=  10;
	calc1491: LREAL :=  10;
	calc1492: LREAL :=  10;
	calc1493: LREAL :=  10;
	calc1494: LREAL :=  10;
	calc1495: LREAL :=  10;
	calc1496: LREAL :=  10;
	calc1497: LREAL :=  10;
	calc1498: LREAL :=  10;
	calc1499: LREAL :=  10;
	calc1500: LREAL :=  10;
	calc1501: LREAL :=  10;
	calc1502: LREAL :=  10;
	calc1503: LREAL :=  10;
	calc1504: LREAL :=  10;
	calc1505: LREAL :=  10;
	calc1506: LREAL :=  10;
	calc1507: LREAL :=  10;
	calc1508: LREAL :=  10;
	calc1509: LREAL :=  10;
	calc1510: LREAL :=  10;
	calc1511: LREAL :=  10;
	calc1512: LREAL :=  10;
	calc1513: LREAL :=  10;
	calc1514: LREAL :=  10;
	calc1515: LREAL :=  10;
	calc1516: LREAL :=  10;
	calc1517: LREAL :=  10;
	calc1518: LREAL :=  10;
	calc1519: LREAL :=  10;
	calc1520: LREAL :=  10;
	calc1521: LREAL :=  10;
	calc1522: LREAL :=  10;
	calc1523: LREAL :=  10;
	calc1524: LREAL :=  10;
	calc1525: LREAL :=  10;
	calc1526: LREAL :=  10;
	calc1527: LREAL :=  10;
	calc1528: LREAL :=  10;
	calc1529: LREAL :=  10;
	calc1530: LREAL :=  10;
	calc1531: LREAL :=  10;
	calc1532: LREAL :=  10;
	calc1533: LREAL :=  10;
	calc1534: LREAL :=  10;
	calc1535: LREAL :=  10;
	calc1536: LREAL :=  10;
	calc1537: LREAL :=  10;
	calc1538: LREAL :=  10;
	calc1539: LREAL :=  10;
	calc1540: LREAL :=  10;
	calc1541: LREAL :=  10;
	calc1542: LREAL :=  10;
	calc1543: LREAL :=  10;
	calc1544: LREAL :=  10;
	calc1545: LREAL :=  10;
	calc1546: LREAL :=  10;
	calc1547: LREAL :=  10;
	calc1548: LREAL :=  10;
	calc1549: LREAL :=  10;
	calc1550: LREAL :=  10;
	calc1551: LREAL :=  10;
	calc1552: LREAL :=  10;
	calc1553: LREAL :=  10;
	calc1554: LREAL :=  10;
	calc1555: LREAL :=  10;
	calc1556: LREAL :=  10;
	calc1557: LREAL :=  10;
	calc1558: LREAL :=  10;
	calc1559: LREAL :=  10;
	calc1560: LREAL :=  10;
	calc1561: LREAL :=  10;
	calc1562: LREAL :=  10;
	calc1563: LREAL :=  10;
	calc1564: LREAL :=  10;
	calc1565: LREAL :=  10;
	calc1566: LREAL :=  10;
	calc1567: LREAL :=  10;
	calc1568: LREAL :=  10;
	calc1569: LREAL :=  10;
	calc1570: LREAL :=  10;
	calc1571: LREAL :=  10;
	calc1572: LREAL :=  10;
	calc1573: LREAL :=  10;
	calc1574: LREAL :=  10;
	calc1575: LREAL :=  10;
	calc1576: LREAL :=  10;
	calc1577: LREAL :=  10;
	calc1578: LREAL :=  10;
	calc1579: LREAL :=  10;
	calc1580: LREAL :=  10;
	calc1581: LREAL :=  10;
	calc1582: LREAL :=  10;
	calc1583: LREAL :=  10;
	calc1584: LREAL :=  10;
	calc1585: LREAL :=  10;
	calc1586: LREAL :=  10;
	calc1587: LREAL :=  10;
	calc1588: LREAL :=  10;
	calc1589: LREAL :=  10;
	calc1590: LREAL :=  10;
	calc1591: LREAL :=  10;
	calc1592: LREAL :=  10;
	calc1593: LREAL :=  10;
	calc1594: LREAL :=  10;
	calc1595: LREAL :=  10;
	calc1596: LREAL :=  10;
	calc1597: LREAL :=  10;
	calc1598: LREAL :=  10;
	calc1599: LREAL :=  10;
	calc1600: LREAL :=  10;
	calc1601: LREAL :=  10;
	calc1602: LREAL :=  10;
	calc1603: LREAL :=  10;
	calc1604: LREAL :=  10;
	calc1605: LREAL :=  10;
	calc1606: LREAL :=  10;
	calc1607: LREAL :=  10;
	calc1608: LREAL :=  10;
	calc1609: LREAL :=  10;
	calc1610: LREAL :=  10;
	calc1611: LREAL :=  10;
	calc1612: LREAL :=  10;
	calc1613: LREAL :=  10;
	calc1614: LREAL :=  10;
	calc1615: LREAL :=  10;
	calc1616: LREAL :=  10;
	calc1617: LREAL :=  10;
	calc1618: LREAL :=  10;
	calc1619: LREAL :=  10;
	calc1620: LREAL :=  10;
	calc1621: LREAL :=  10;
	calc1622: LREAL :=  10;
	calc1623: LREAL :=  10;
	calc1624: LREAL :=  10;
	calc1625: LREAL :=  10;
	calc1626: LREAL :=  10;
	calc1627: LREAL :=  10;
	calc1628: LREAL :=  10;
	calc1629: LREAL :=  10;
	calc1630: LREAL :=  10;
	calc1631: LREAL :=  10;
	calc1632: LREAL :=  10;
	calc1633: LREAL :=  10;
	calc1634: LREAL :=  10;
	calc1635: LREAL :=  10;
	calc1636: LREAL :=  10;
	calc1637: LREAL :=  10;
	calc1638: LREAL :=  10;
	calc1639: LREAL :=  10;
	calc1640: LREAL :=  10;
	calc1641: LREAL :=  10;
	calc1642: LREAL :=  10;
	calc1643: LREAL :=  10;
	calc1644: LREAL :=  10;
	calc1645: LREAL :=  10;
	calc1646: LREAL :=  10;
	calc1647: LREAL :=  10;
	calc1648: LREAL :=  10;
	calc1649: LREAL :=  10;
	calc1650: LREAL :=  10;
	calc1651: LREAL :=  10;
	calc1652: LREAL :=  10;
	calc1653: LREAL :=  10;
	calc1654: LREAL :=  10;
	calc1655: LREAL :=  10;
	calc1656: LREAL :=  10;
	calc1657: LREAL :=  10;
	calc1658: LREAL :=  10;
	calc1659: LREAL :=  10;
	calc1660: LREAL :=  10;
	calc1661: LREAL :=  10;
	calc1662: LREAL :=  10;
	calc1663: LREAL :=  10;
	calc1664: LREAL :=  10;
	calc1665: LREAL :=  10;
	calc1666: LREAL :=  10;
	calc1667: LREAL :=  10;
	calc1668: LREAL :=  10;
	calc1669: LREAL :=  10;
	calc1670: LREAL :=  10;
	calc1671: LREAL :=  10;
	calc1672: LREAL :=  10;
	calc1673: LREAL :=  10;
	calc1674: LREAL :=  10;
	calc1675: LREAL :=  10;
	calc1676: LREAL :=  10;
	calc1677: LREAL :=  10;
	calc1678: LREAL :=  10;
	calc1679: LREAL :=  10;
	calc1680: LREAL :=  10;
	calc1681: LREAL :=  10;
	calc1682: LREAL :=  10;
	calc1683: LREAL :=  10;
	calc1684: LREAL :=  10;
	calc1685: LREAL :=  10;
	calc1686: LREAL :=  10;
	calc1687: LREAL :=  10;
	calc1688: LREAL :=  10;
	calc1689: LREAL :=  10;
	calc1690: LREAL :=  10;
	calc1691: LREAL :=  10;
	calc1692: LREAL :=  10;
	calc1693: LREAL :=  10;
	calc1694: LREAL :=  10;
	calc1695: LREAL :=  10;
	calc1696: LREAL :=  10;
	calc1697: LREAL :=  10;
	calc1698: LREAL :=  10;
	calc1699: LREAL :=  10;
	calc1700: LREAL :=  10;
	calc1701: LREAL :=  10;
	calc1702: LREAL :=  10;
	calc1703: LREAL :=  10;
	calc1704: LREAL :=  10;
	calc1705: LREAL :=  10;
	calc1706: LREAL :=  10;
	calc1707: LREAL :=  10;
	calc1708: LREAL :=  10;
	calc1709: LREAL :=  10;
	calc1710: LREAL :=  10;
	calc1711: LREAL :=  10;
	calc1712: LREAL :=  10;
	calc1713: LREAL :=  10;
	calc1714: LREAL :=  10;
	calc1715: LREAL :=  10;
	calc1716: LREAL :=  10;
	calc1717: LREAL :=  10;
	calc1718: LREAL :=  10;
	calc1719: LREAL :=  10;
	calc1720: LREAL :=  10;
	calc1721: LREAL :=  10;
	calc1722: LREAL :=  10;
	calc1723: LREAL :=  10;
	calc1724: LREAL :=  10;
	calc1725: LREAL :=  10;
	calc1726: LREAL :=  10;
	calc1727: LREAL :=  10;
	calc1728: LREAL :=  10;
	calc1729: LREAL :=  10;
	calc1730: LREAL :=  10;
	calc1731: LREAL :=  10;
	calc1732: LREAL :=  10;
	calc1733: LREAL :=  10;
	calc1734: LREAL :=  10;
	calc1735: LREAL :=  10;
	calc1736: LREAL :=  10;
	calc1737: LREAL :=  10;
	calc1738: LREAL :=  10;
	calc1739: LREAL :=  10;
	calc1740: LREAL :=  10;
	calc1741: LREAL :=  10;
	calc1742: LREAL :=  10;
	calc1743: LREAL :=  10;
	calc1744: LREAL :=  10;
	calc1745: LREAL :=  10;
	calc1746: LREAL :=  10;
	calc1747: LREAL :=  10;
	calc1748: LREAL :=  10;
	calc1749: LREAL :=  10;
	calc1750: LREAL :=  10;
	calc1751: LREAL :=  10;
	calc1752: LREAL :=  10;
	calc1753: LREAL :=  10;
	calc1754: LREAL :=  10;
	calc1755: LREAL :=  10;
	calc1756: LREAL :=  10;
	calc1757: LREAL :=  10;
	calc1758: LREAL :=  10;
	calc1759: LREAL :=  10;
	calc1760: LREAL :=  10;
	calc1761: LREAL :=  10;
	calc1762: LREAL :=  10;
	calc1763: LREAL :=  10;
	calc1764: LREAL :=  10;
	calc1765: LREAL :=  10;
	calc1766: LREAL :=  10;
	calc1767: LREAL :=  10;
	calc1768: LREAL :=  10;
	calc1769: LREAL :=  10;
	calc1770: LREAL :=  10;
	calc1771: LREAL :=  10;
	calc1772: LREAL :=  10;
	calc1773: LREAL :=  10;
	calc1774: LREAL :=  10;
	calc1775: LREAL :=  10;
	calc1776: LREAL :=  10;
	calc1777: LREAL :=  10;
	calc1778: LREAL :=  10;
	calc1779: LREAL :=  10;
	calc1780: LREAL :=  10;
	calc1781: LREAL :=  10;
	calc1782: LREAL :=  10;
	calc1783: LREAL :=  10;
	calc1784: LREAL :=  10;
	calc1785: LREAL :=  10;
	calc1786: LREAL :=  10;
	calc1787: LREAL :=  10;
	calc1788: LREAL :=  10;
	calc1789: LREAL :=  10;
	calc1790: LREAL :=  10;
	calc1791: LREAL :=  10;
	calc1792: LREAL :=  10;
	calc1793: LREAL :=  10;
	calc1794: LREAL :=  10;
	calc1795: LREAL :=  10;
	calc1796: LREAL :=  10;
	calc1797: LREAL :=  10;
	calc1798: LREAL :=  10;
	calc1799: LREAL :=  10;
	calc1800: LREAL :=  10;
	calc1801: LREAL :=  10;
	calc1802: LREAL :=  10;
	calc1803: LREAL :=  10;
	calc1804: LREAL :=  10;
	calc1805: LREAL :=  10;
	calc1806: LREAL :=  10;
	calc1807: LREAL :=  10;
	calc1808: LREAL :=  10;
	calc1809: LREAL :=  10;
	calc1810: LREAL :=  10;
	calc1811: LREAL :=  10;
	calc1812: LREAL :=  10;
	calc1813: LREAL :=  10;
	calc1814: LREAL :=  10;
	calc1815: LREAL :=  10;
	calc1816: LREAL :=  10;
	calc1817: LREAL :=  10;
	calc1818: LREAL :=  10;
	calc1819: LREAL :=  10;
	calc1820: LREAL :=  10;
	calc1821: LREAL :=  10;
	calc1822: LREAL :=  10;
	calc1823: LREAL :=  10;
	calc1824: LREAL :=  10;
	calc1825: LREAL :=  10;
	calc1826: LREAL :=  10;
	calc1827: LREAL :=  10;
	calc1828: LREAL :=  10;
	calc1829: LREAL :=  10;
	calc1830: LREAL :=  10;
	calc1831: LREAL :=  10;
	calc1832: LREAL :=  10;
	calc1833: LREAL :=  10;
	calc1834: LREAL :=  10;
	calc1835: LREAL :=  10;
	calc1836: LREAL :=  10;
	calc1837: LREAL :=  10;
	calc1838: LREAL :=  10;
	calc1839: LREAL :=  10;
	calc1840: LREAL :=  10;
	calc1841: LREAL :=  10;
	calc1842: LREAL :=  10;
	calc1843: LREAL :=  10;
	calc1844: LREAL :=  10;
	calc1845: LREAL :=  10;
	calc1846: LREAL :=  10;
	calc1847: LREAL :=  10;
	calc1848: LREAL :=  10;
	calc1849: LREAL :=  10;
	calc1850: LREAL :=  10;
	calc1851: LREAL :=  10;
	calc1852: LREAL :=  10;
	calc1853: LREAL :=  10;
	calc1854: LREAL :=  10;
	calc1855: LREAL :=  10;
	calc1856: LREAL :=  10;
	calc1857: LREAL :=  10;
	calc1858: LREAL :=  10;
	calc1859: LREAL :=  10;
	calc1860: LREAL :=  10;
	calc1861: LREAL :=  10;
	calc1862: LREAL :=  10;
	calc1863: LREAL :=  10;
	calc1864: LREAL :=  10;
	calc1865: LREAL :=  10;
	calc1866: LREAL :=  10;
	calc1867: LREAL :=  10;
	calc1868: LREAL :=  10;
	calc1869: LREAL :=  10;
	calc1870: LREAL :=  10;
	calc1871: LREAL :=  10;
	calc1872: LREAL :=  10;
	calc1873: LREAL :=  10;
	calc1874: LREAL :=  10;
	calc1875: LREAL :=  10;
	calc1876: LREAL :=  10;
	calc1877: LREAL :=  10;
	calc1878: LREAL :=  10;
	calc1879: LREAL :=  10;
	calc1880: LREAL :=  10;
	calc1881: LREAL :=  10;
	calc1882: LREAL :=  10;
	calc1883: LREAL :=  10;
	calc1884: LREAL :=  10;
	calc1885: LREAL :=  10;
	calc1886: LREAL :=  10;
	calc1887: LREAL :=  10;
	calc1888: LREAL :=  10;
	calc1889: LREAL :=  10;
	calc1890: LREAL :=  10;
	calc1891: LREAL :=  10;
	calc1892: LREAL :=  10;
	calc1893: LREAL :=  10;
	calc1894: LREAL :=  10;
	calc1895: LREAL :=  10;
	calc1896: LREAL :=  10;
	calc1897: LREAL :=  10;
	calc1898: LREAL :=  10;
	calc1899: LREAL :=  10;
	calc1900: LREAL :=  10;
	calc1901: LREAL :=  10;
	calc1902: LREAL :=  10;
	calc1903: LREAL :=  10;
	calc1904: LREAL :=  10;
	calc1905: LREAL :=  10;
	calc1906: LREAL :=  10;
	calc1907: LREAL :=  10;
	calc1908: LREAL :=  10;
	calc1909: LREAL :=  10;
	calc1910: LREAL :=  10;
	calc1911: LREAL :=  10;
	calc1912: LREAL :=  10;
	calc1913: LREAL :=  10;
	calc1914: LREAL :=  10;
	calc1915: LREAL :=  10;
	calc1916: LREAL :=  10;
	calc1917: LREAL :=  10;
	calc1918: LREAL :=  10;
	calc1919: LREAL :=  10;
	calc1920: LREAL :=  10;
	calc1921: LREAL :=  10;
	calc1922: LREAL :=  10;
	calc1923: LREAL :=  10;
	calc1924: LREAL :=  10;
	calc1925: LREAL :=  10;
	calc1926: LREAL :=  10;
	calc1927: LREAL :=  10;
	calc1928: LREAL :=  10;
	calc1929: LREAL :=  10;
	calc1930: LREAL :=  10;
	calc1931: LREAL :=  10;
	calc1932: LREAL :=  10;
	calc1933: LREAL :=  10;
	calc1934: LREAL :=  10;
	calc1935: LREAL :=  10;
	calc1936: LREAL :=  10;
	calc1937: LREAL :=  10;
	calc1938: LREAL :=  10;
	calc1939: LREAL :=  10;
	calc1940: LREAL :=  10;
	calc1941: LREAL :=  10;
	calc1942: LREAL :=  10;
	calc1943: LREAL :=  10;
	calc1944: LREAL :=  10;
	calc1945: LREAL :=  10;
	calc1946: LREAL :=  10;
	calc1947: LREAL :=  10;
	calc1948: LREAL :=  10;
	calc1949: LREAL :=  10;
	calc1950: LREAL :=  10;
	calc1951: LREAL :=  10;
	calc1952: LREAL :=  10;
	calc1953: LREAL :=  10;
	calc1954: LREAL :=  10;
	calc1955: LREAL :=  10;
	calc1956: LREAL :=  10;
	calc1957: LREAL :=  10;
	calc1958: LREAL :=  10;
	calc1959: LREAL :=  10;
	calc1960: LREAL :=  10;
	calc1961: LREAL :=  10;
	calc1962: LREAL :=  10;
	calc1963: LREAL :=  10;
	calc1964: LREAL :=  10;
	calc1965: LREAL :=  10;
	calc1966: LREAL :=  10;
	calc1967: LREAL :=  10;
	calc1968: LREAL :=  10;
	calc1969: LREAL :=  10;
	calc1970: LREAL :=  10;
	calc1971: LREAL :=  10;
	calc1972: LREAL :=  10;
	calc1973: LREAL :=  10;
	calc1974: LREAL :=  10;
	calc1975: LREAL :=  10;
	calc1976: LREAL :=  10;
	calc1977: LREAL :=  10;
	calc1978: LREAL :=  10;
	calc1979: LREAL :=  10;
	calc1980: LREAL :=  10;
	calc1981: LREAL :=  10;
	calc1982: LREAL :=  10;
	calc1983: LREAL :=  10;
	calc1984: LREAL :=  10;
	calc1985: LREAL :=  10;
	calc1986: LREAL :=  10;
	calc1987: LREAL :=  10;
	calc1988: LREAL :=  10;
	calc1989: LREAL :=  10;
	calc1990: LREAL :=  10;
	calc1991: LREAL :=  10;
	calc1992: LREAL :=  10;
	calc1993: LREAL :=  10;
	calc1994: LREAL :=  10;
	calc1995: LREAL :=  10;
	calc1996: LREAL :=  10;
	calc1997: LREAL :=  10;
	calc1998: LREAL :=  10;
	calc1999: LREAL :=  10;
	calc2000: LREAL :=  10;
	calc2001: LREAL :=  10;
	calc2002: LREAL :=  10;
	calc2003: LREAL :=  10;
	calc2004: LREAL :=  10;
	calc2005: LREAL :=  10;
	calc2006: LREAL :=  10;
	calc2007: LREAL :=  10;
	calc2008: LREAL :=  10;
	calc2009: LREAL :=  10;
	calc2010: LREAL :=  10;
	calc2011: LREAL :=  10;
	calc2012: LREAL :=  10;
	calc2013: LREAL :=  10;
	calc2014: LREAL :=  10;
	calc2015: LREAL :=  10;
	calc2016: LREAL :=  10;
	calc2017: LREAL :=  10;
	calc2018: LREAL :=  10;
	calc2019: LREAL :=  10;
	calc2020: LREAL :=  10;
	calc2021: LREAL :=  10;
	calc2022: LREAL :=  10;
	calc2023: LREAL :=  10;
	calc2024: LREAL :=  10;
	calc2025: LREAL :=  10;
	calc2026: LREAL :=  10;
	calc2027: LREAL :=  10;
	calc2028: LREAL :=  10;
	calc2029: LREAL :=  10;
	calc2030: LREAL :=  10;
	calc2031: LREAL :=  10;
	calc2032: LREAL :=  10;
	calc2033: LREAL :=  10;
	calc2034: LREAL :=  10;
	calc2035: LREAL :=  10;
	calc2036: LREAL :=  10;
	calc2037: LREAL :=  10;
	calc2038: LREAL :=  10;
	calc2039: LREAL :=  10;
	calc2040: LREAL :=  10;
	calc2041: LREAL :=  10;
	calc2042: LREAL :=  10;
	calc2043: LREAL :=  10;
	calc2044: LREAL :=  10;
	calc2045: LREAL :=  10;
	calc2046: LREAL :=  10;
	calc2047: LREAL :=  10;
	calc2048: LREAL :=  10;
	calc2049: LREAL :=  10;
	calc2050: LREAL :=  10;
	calc2051: LREAL :=  10;
	calc2052: LREAL :=  10;
	calc2053: LREAL :=  10;
	calc2054: LREAL :=  10;
	calc2055: LREAL :=  10;
	calc2056: LREAL :=  10;
	calc2057: LREAL :=  10;
	calc2058: LREAL :=  10;
	calc2059: LREAL :=  10;
	calc2060: LREAL :=  10;
	calc2061: LREAL :=  10;
	calc2062: LREAL :=  10;
	calc2063: LREAL :=  10;
	calc2064: LREAL :=  10;
	calc2065: LREAL :=  10;
	calc2066: LREAL :=  10;
	calc2067: LREAL :=  10;
	calc2068: LREAL :=  10;
	calc2069: LREAL :=  10;
	calc2070: LREAL :=  10;
	calc2071: LREAL :=  10;
	calc2072: LREAL :=  10;
	calc2073: LREAL :=  10;
	calc2074: LREAL :=  10;
	calc2075: LREAL :=  10;
	calc2076: LREAL :=  10;
	calc2077: LREAL :=  10;
	calc2078: LREAL :=  10;
	calc2079: LREAL :=  10;
	calc2080: LREAL :=  10;
	calc2081: LREAL :=  10;
	calc2082: LREAL :=  10;
	calc2083: LREAL :=  10;
	calc2084: LREAL :=  10;
	calc2085: LREAL :=  10;
	calc2086: LREAL :=  10;
	calc2087: LREAL :=  10;
	calc2088: LREAL :=  10;
	calc2089: LREAL :=  10;
	calc2090: LREAL :=  10;
	calc2091: LREAL :=  10;
	calc2092: LREAL :=  10;
	calc2093: LREAL :=  10;
	calc2094: LREAL :=  10;
	calc2095: LREAL :=  10;
	calc2096: LREAL :=  10;
	calc2097: LREAL :=  10;
	calc2098: LREAL :=  10;
	calc2099: LREAL :=  10;
	calc2100: LREAL :=  10;
	calc2101: LREAL :=  10;
	calc2102: LREAL :=  10;
	calc2103: LREAL :=  10;
	calc2104: LREAL :=  10;
	calc2105: LREAL :=  10;
	calc2106: LREAL :=  10;
	calc2107: LREAL :=  10;
	calc2108: LREAL :=  10;
	calc2109: LREAL :=  10;
	calc2110: LREAL :=  10;
	calc2111: LREAL :=  10;
	calc2112: LREAL :=  10;
	calc2113: LREAL :=  10;
	calc2114: LREAL :=  10;
	calc2115: LREAL :=  10;
	calc2116: LREAL :=  10;
	calc2117: LREAL :=  10;
	calc2118: LREAL :=  10;
	calc2119: LREAL :=  10;
	calc2120: LREAL :=  10;
	calc2121: LREAL :=  10;
	calc2122: LREAL :=  10;
	calc2123: LREAL :=  10;
	calc2124: LREAL :=  10;
	calc2125: LREAL :=  10;
	calc2126: LREAL :=  10;
	calc2127: LREAL :=  10;
	calc2128: LREAL :=  10;
	calc2129: LREAL :=  10;
	calc2130: LREAL :=  10;
	calc2131: LREAL :=  10;
	calc2132: LREAL :=  10;
	calc2133: LREAL :=  10;
	calc2134: LREAL :=  10;
	calc2135: LREAL :=  10;
	calc2136: LREAL :=  10;
	calc2137: LREAL :=  10;
	calc2138: LREAL :=  10;
	calc2139: LREAL :=  10;
	calc2140: LREAL :=  10;
	calc2141: LREAL :=  10;
	calc2142: LREAL :=  10;
	calc2143: LREAL :=  10;
	calc2144: LREAL :=  10;
	calc2145: LREAL :=  10;
	calc2146: LREAL :=  10;
	calc2147: LREAL :=  10;
	calc2148: LREAL :=  10;
	calc2149: LREAL :=  10;
	calc2150: LREAL :=  10;
	calc2151: LREAL :=  10;
	calc2152: LREAL :=  10;
	calc2153: LREAL :=  10;
	calc2154: LREAL :=  10;
	calc2155: LREAL :=  10;
	calc2156: LREAL :=  10;
	calc2157: LREAL :=  10;
	calc2158: LREAL :=  10;
	calc2159: LREAL :=  10;
	calc2160: LREAL :=  10;
	calc2161: LREAL :=  10;
	calc2162: LREAL :=  10;
	calc2163: LREAL :=  10;
	calc2164: LREAL :=  10;
	calc2165: LREAL :=  10;
	calc2166: LREAL :=  10;
	calc2167: LREAL :=  10;
	calc2168: LREAL :=  10;
	calc2169: LREAL :=  10;
	calc2170: LREAL :=  10;
	calc2171: LREAL :=  10;
	calc2172: LREAL :=  10;
	calc2173: LREAL :=  10;
	calc2174: LREAL :=  10;
	calc2175: LREAL :=  10;
	calc2176: LREAL :=  10;
	calc2177: LREAL :=  10;
	calc2178: LREAL :=  10;
	calc2179: LREAL :=  10;
	calc2180: LREAL :=  10;
	calc2181: LREAL :=  10;
	calc2182: LREAL :=  10;
	calc2183: LREAL :=  10;
	calc2184: LREAL :=  10;
	calc2185: LREAL :=  10;
	calc2186: LREAL :=  10;
	calc2187: LREAL :=  10;
	calc2188: LREAL :=  10;
	calc2189: LREAL :=  10;
	calc2190: LREAL :=  10;
	calc2191: LREAL :=  10;
	calc2192: LREAL :=  10;
	calc2193: LREAL :=  10;
	calc2194: LREAL :=  10;
	calc2195: LREAL :=  10;
	calc2196: LREAL :=  10;
	calc2197: LREAL :=  10;
	calc2198: LREAL :=  10;
	calc2199: LREAL :=  10;
	calc2200: LREAL :=  10;
	calc2201: LREAL :=  10;
	calc2202: LREAL :=  10;
	calc2203: LREAL :=  10;
	calc2204: LREAL :=  10;
	calc2205: LREAL :=  10;
	calc2206: LREAL :=  10;
	calc2207: LREAL :=  10;
	calc2208: LREAL :=  10;
	calc2209: LREAL :=  10;
	calc2210: LREAL :=  10;
	calc2211: LREAL :=  10;
	calc2212: LREAL :=  10;
	calc2213: LREAL :=  10;
	calc2214: LREAL :=  10;
	calc2215: LREAL :=  10;
	calc2216: LREAL :=  10;
	calc2217: LREAL :=  10;
	calc2218: LREAL :=  10;
	calc2219: LREAL :=  10;
	calc2220: LREAL :=  10;
	calc2221: LREAL :=  10;
	calc2222: LREAL :=  10;
	calc2223: LREAL :=  10;
	calc2224: LREAL :=  10;
	calc2225: LREAL :=  10;
	calc2226: LREAL :=  10;
	calc2227: LREAL :=  10;
	calc2228: LREAL :=  10;
	calc2229: LREAL :=  10;
	calc2230: LREAL :=  10;
	calc2231: LREAL :=  10;
	calc2232: LREAL :=  10;
	calc2233: LREAL :=  10;
	calc2234: LREAL :=  10;
	calc2235: LREAL :=  10;
	calc2236: LREAL :=  10;
	calc2237: LREAL :=  10;
	calc2238: LREAL :=  10;
	calc2239: LREAL :=  10;
	calc2240: LREAL :=  10;
	calc2241: LREAL :=  10;
	calc2242: LREAL :=  10;
	calc2243: LREAL :=  10;
	calc2244: LREAL :=  10;
	calc2245: LREAL :=  10;
	calc2246: LREAL :=  10;
	calc2247: LREAL :=  10;
	calc2248: LREAL :=  10;
	calc2249: LREAL :=  10;
	calc2250: LREAL :=  10;
	calc2251: LREAL :=  10;
	calc2252: LREAL :=  10;
	calc2253: LREAL :=  10;
	calc2254: LREAL :=  10;
	calc2255: LREAL :=  10;
	calc2256: LREAL :=  10;
	calc2257: LREAL :=  10;
	calc2258: LREAL :=  10;
	calc2259: LREAL :=  10;
	calc2260: LREAL :=  10;
	calc2261: LREAL :=  10;
	calc2262: LREAL :=  10;
	calc2263: LREAL :=  10;
	calc2264: LREAL :=  10;
	calc2265: LREAL :=  10;
	calc2266: LREAL :=  10;
	calc2267: LREAL :=  10;
	calc2268: LREAL :=  10;
	calc2269: LREAL :=  10;
	calc2270: LREAL :=  10;
	calc2271: LREAL :=  10;
	calc2272: LREAL :=  10;
	calc2273: LREAL :=  10;
	calc2274: LREAL :=  10;
	calc2275: LREAL :=  10;
	calc2276: LREAL :=  10;
	calc2277: LREAL :=  10;
	calc2278: LREAL :=  10;
	calc2279: LREAL :=  10;
	calc2280: LREAL :=  10;
	calc2281: LREAL :=  10;
	calc2282: LREAL :=  10;
	calc2283: LREAL :=  10;
	calc2284: LREAL :=  10;
	calc2285: LREAL :=  10;
	calc2286: LREAL :=  10;
	calc2287: LREAL :=  10;
	calc2288: LREAL :=  10;
	calc2289: LREAL :=  10;
	calc2290: LREAL :=  10;
	calc2291: LREAL :=  10;
	calc2292: LREAL :=  10;
	calc2293: LREAL :=  10;
	calc2294: LREAL :=  10;
	calc2295: LREAL :=  10;
	calc2296: LREAL :=  10;
	calc2297: LREAL :=  10;
	calc2298: LREAL :=  10;
	calc2299: LREAL :=  10;
	calc2300: LREAL :=  10;
	calc2301: LREAL :=  10;
	calc2302: LREAL :=  10;
	calc2303: LREAL :=  10;
	calc2304: LREAL :=  10;
	calc2305: LREAL :=  10;
	calc2306: LREAL :=  10;
	calc2307: LREAL :=  10;
	calc2308: LREAL :=  10;
	calc2309: LREAL :=  10;
	calc2310: LREAL :=  10;
	calc2311: LREAL :=  10;
	calc2312: LREAL :=  10;
	calc2313: LREAL :=  10;
	calc2314: LREAL :=  10;
	calc2315: LREAL :=  10;
	calc2316: LREAL :=  10;
	calc2317: LREAL :=  10;
	calc2318: LREAL :=  10;
	calc2319: LREAL :=  10;
	calc2320: LREAL :=  10;
	calc2321: LREAL :=  10;
	calc2322: LREAL :=  10;
	calc2323: LREAL :=  10;
	calc2324: LREAL :=  10;
	calc2325: LREAL :=  10;
	calc2326: LREAL :=  10;
	calc2327: LREAL :=  10;
	calc2328: LREAL :=  10;
	calc2329: LREAL :=  10;
	calc2330: LREAL :=  10;
	calc2331: LREAL :=  10;
	calc2332: LREAL :=  10;
	calc2333: LREAL :=  10;
	calc2334: LREAL :=  10;
	calc2335: LREAL :=  10;
	calc2336: LREAL :=  10;
	calc2337: LREAL :=  10;
	calc2338: LREAL :=  10;
	calc2339: LREAL :=  10;
	calc2340: LREAL :=  10;
	calc2341: LREAL :=  10;
	calc2342: LREAL :=  10;
	calc2343: LREAL :=  10;
	calc2344: LREAL :=  10;
	calc2345: LREAL :=  10;
	calc2346: LREAL :=  10;
	calc2347: LREAL :=  10;
	calc2348: LREAL :=  10;
	calc2349: LREAL :=  10;
	calc2350: LREAL :=  10;
	calc2351: LREAL :=  10;
	calc2352: LREAL :=  10;
	calc2353: LREAL :=  10;
	calc2354: LREAL :=  10;
	calc2355: LREAL :=  10;
	calc2356: LREAL :=  10;
	calc2357: LREAL :=  10;
	calc2358: LREAL :=  10;
	calc2359: LREAL :=  10;
	calc2360: LREAL :=  10;
	calc2361: LREAL :=  10;
	calc2362: LREAL :=  10;
	calc2363: LREAL :=  10;
	calc2364: LREAL :=  10;
	calc2365: LREAL :=  10;
	calc2366: LREAL :=  10;
	calc2367: LREAL :=  10;
	calc2368: LREAL :=  10;
	calc2369: LREAL :=  10;
	calc2370: LREAL :=  10;
	calc2371: LREAL :=  10;
	calc2372: LREAL :=  10;
	calc2373: LREAL :=  10;
	calc2374: LREAL :=  10;
	calc2375: LREAL :=  10;
	calc2376: LREAL :=  10;
	calc2377: LREAL :=  10;
	calc2378: LREAL :=  10;
	calc2379: LREAL :=  10;
	calc2380: LREAL :=  10;
	calc2381: LREAL :=  10;
	calc2382: LREAL :=  10;
	calc2383: LREAL :=  10;
	calc2384: LREAL :=  10;
	calc2385: LREAL :=  10;
	calc2386: LREAL :=  10;
	calc2387: LREAL :=  10;
	calc2388: LREAL :=  10;
	calc2389: LREAL :=  10;
	calc2390: LREAL :=  10;
	calc2391: LREAL :=  10;
	calc2392: LREAL :=  10;
	calc2393: LREAL :=  10;
	calc2394: LREAL :=  10;
	calc2395: LREAL :=  10;
	calc2396: LREAL :=  10;
	calc2397: LREAL :=  10;
	calc2398: LREAL :=  10;
	calc2399: LREAL :=  10;
	calc2400: LREAL :=  10;
	calc2401: LREAL :=  10;
	calc2402: LREAL :=  10;
	calc2403: LREAL :=  10;
	calc2404: LREAL :=  10;
	calc2405: LREAL :=  10;
	calc2406: LREAL :=  10;
	calc2407: LREAL :=  10;
	calc2408: LREAL :=  10;
	calc2409: LREAL :=  10;
	calc2410: LREAL :=  10;
	calc2411: LREAL :=  10;
	calc2412: LREAL :=  10;
	calc2413: LREAL :=  10;
	calc2414: LREAL :=  10;
	calc2415: LREAL :=  10;
	calc2416: LREAL :=  10;
	calc2417: LREAL :=  10;
	calc2418: LREAL :=  10;
	calc2419: LREAL :=  10;
	calc2420: LREAL :=  10;
	calc2421: LREAL :=  10;
	calc2422: LREAL :=  10;
	calc2423: LREAL :=  10;
	calc2424: LREAL :=  10;
	calc2425: LREAL :=  10;
	calc2426: LREAL :=  10;
	calc2427: LREAL :=  10;
	calc2428: LREAL :=  10;
	calc2429: LREAL :=  10;
	calc2430: LREAL :=  10;
	calc2431: LREAL :=  10;
	calc2432: LREAL :=  10;
	calc2433: LREAL :=  10;
	calc2434: LREAL :=  10;
	calc2435: LREAL :=  10;
	calc2436: LREAL :=  10;
	calc2437: LREAL :=  10;
	calc2438: LREAL :=  10;
	calc2439: LREAL :=  10;
	calc2440: LREAL :=  10;
	calc2441: LREAL :=  10;
	calc2442: LREAL :=  10;
	calc2443: LREAL :=  10;
	calc2444: LREAL :=  10;
	calc2445: LREAL :=  10;
	calc2446: LREAL :=  10;
	calc2447: LREAL :=  10;
	calc2448: LREAL :=  10;
	calc2449: LREAL :=  10;
	calc2450: LREAL :=  10;
	calc2451: LREAL :=  10;
	calc2452: LREAL :=  10;
	calc2453: LREAL :=  10;
	calc2454: LREAL :=  10;
	calc2455: LREAL :=  10;
	calc2456: LREAL :=  10;
	calc2457: LREAL :=  10;
	calc2458: LREAL :=  10;
	calc2459: LREAL :=  10;
	calc2460: LREAL :=  10;
	calc2461: LREAL :=  10;
	calc2462: LREAL :=  10;
	calc2463: LREAL :=  10;
	calc2464: LREAL :=  10;
	calc2465: LREAL :=  10;
	calc2466: LREAL :=  10;
	calc2467: LREAL :=  10;
	calc2468: LREAL :=  10;
	calc2469: LREAL :=  10;
	calc2470: LREAL :=  10;
	calc2471: LREAL :=  10;
	calc2472: LREAL :=  10;
	calc2473: LREAL :=  10;
	calc2474: LREAL :=  10;
	calc2475: LREAL :=  10;
	calc2476: LREAL :=  10;
	calc2477: LREAL :=  10;
	calc2478: LREAL :=  10;
	calc2479: LREAL :=  10;
	calc2480: LREAL :=  10;
	calc2481: LREAL :=  10;
	calc2482: LREAL :=  10;
	calc2483: LREAL :=  10;
	calc2484: LREAL :=  10;
	calc2485: LREAL :=  10;
	calc2486: LREAL :=  10;
	calc2487: LREAL :=  10;
	calc2488: LREAL :=  10;
	calc2489: LREAL :=  10;
	calc2490: LREAL :=  10;
	calc2491: LREAL :=  10;
	calc2492: LREAL :=  10;
	calc2493: LREAL :=  10;
	calc2494: LREAL :=  10;
	calc2495: LREAL :=  10;
	calc2496: LREAL :=  10;
	calc2497: LREAL :=  10;
	calc2498: LREAL :=  10;
	calc2499: LREAL :=  10;
	calc2500: LREAL :=  10;
	calc2501: LREAL :=  10;
	calc2502: LREAL :=  10;
	calc2503: LREAL :=  10;
	calc2504: LREAL :=  10;
	calc2505: LREAL :=  10;
	calc2506: LREAL :=  10;
	calc2507: LREAL :=  10;
	calc2508: LREAL :=  10;
	calc2509: LREAL :=  10;
	calc2510: LREAL :=  10;
	calc2511: LREAL :=  10;
	calc2512: LREAL :=  10;
	calc2513: LREAL :=  10;
	calc2514: LREAL :=  10;
	calc2515: LREAL :=  10;
	calc2516: LREAL :=  10;
	calc2517: LREAL :=  10;
	calc2518: LREAL :=  10;
	calc2519: LREAL :=  10;
	calc2520: LREAL :=  10;
	calc2521: LREAL :=  10;
	calc2522: LREAL :=  10;
	calc2523: LREAL :=  10;
	calc2524: LREAL :=  10;
	calc2525: LREAL :=  10;
	calc2526: LREAL :=  10;
	calc2527: LREAL :=  10;
	calc2528: LREAL :=  10;
	calc2529: LREAL :=  10;
	calc2530: LREAL :=  10;
	calc2531: LREAL :=  10;
	calc2532: LREAL :=  10;
	calc2533: LREAL :=  10;
	calc2534: LREAL :=  10;
	calc2535: LREAL :=  10;
	calc2536: LREAL :=  10;
	calc2537: LREAL :=  10;
	calc2538: LREAL :=  10;
	calc2539: LREAL :=  10;
	calc2540: LREAL :=  10;
	calc2541: LREAL :=  10;
	calc2542: LREAL :=  10;
	calc2543: LREAL :=  10;
	calc2544: LREAL :=  10;
	calc2545: LREAL :=  10;
	calc2546: LREAL :=  10;
	calc2547: LREAL :=  10;
	calc2548: LREAL :=  10;
	calc2549: LREAL :=  10;
	calc2550: LREAL :=  10;
	calc2551: LREAL :=  10;
	calc2552: LREAL :=  10;
	calc2553: LREAL :=  10;
	calc2554: LREAL :=  10;
	calc2555: LREAL :=  10;
	calc2556: LREAL :=  10;
	calc2557: LREAL :=  10;
	calc2558: LREAL :=  10;
	calc2559: LREAL :=  10;
	calc2560: LREAL :=  10;
	calc2561: LREAL :=  10;
	calc2562: LREAL :=  10;
	calc2563: LREAL :=  10;
	calc2564: LREAL :=  10;
	calc2565: LREAL :=  10;
	calc2566: LREAL :=  10;
	calc2567: LREAL :=  10;
	calc2568: LREAL :=  10;
	calc2569: LREAL :=  10;
	calc2570: LREAL :=  10;
	calc2571: LREAL :=  10;
	calc2572: LREAL :=  10;
	calc2573: LREAL :=  10;
	calc2574: LREAL :=  10;
	calc2575: LREAL :=  10;
	calc2576: LREAL :=  10;
	calc2577: LREAL :=  10;
	calc2578: LREAL :=  10;
	calc2579: LREAL :=  10;
	calc2580: LREAL :=  10;
	calc2581: LREAL :=  10;
	calc2582: LREAL :=  10;
	calc2583: LREAL :=  10;
	calc2584: LREAL :=  10;
	calc2585: LREAL :=  10;
	calc2586: LREAL :=  10;
	calc2587: LREAL :=  10;
	calc2588: LREAL :=  10;
	calc2589: LREAL :=  10;
	calc2590: LREAL :=  10;
	calc2591: LREAL :=  10;
	calc2592: LREAL :=  10;
	calc2593: LREAL :=  10;
	calc2594: LREAL :=  10;
	calc2595: LREAL :=  10;
	calc2596: LREAL :=  10;
	calc2597: LREAL :=  10;
	calc2598: LREAL :=  10;
	calc2599: LREAL :=  10;
	calc2600: LREAL :=  10;
	calc2601: LREAL :=  10;
	calc2602: LREAL :=  10;
	calc2603: LREAL :=  10;
	calc2604: LREAL :=  10;
	calc2605: LREAL :=  10;
	calc2606: LREAL :=  10;
	calc2607: LREAL :=  10;
	calc2608: LREAL :=  10;
	calc2609: LREAL :=  10;
	calc2610: LREAL :=  10;
	calc2611: LREAL :=  10;
	calc2612: LREAL :=  10;
	calc2613: LREAL :=  10;
	calc2614: LREAL :=  10;
	calc2615: LREAL :=  10;
	calc2616: LREAL :=  10;
	calc2617: LREAL :=  10;
	calc2618: LREAL :=  10;
	calc2619: LREAL :=  10;
	calc2620: LREAL :=  10;
	calc2621: LREAL :=  10;
	calc2622: LREAL :=  10;
	calc2623: LREAL :=  10;
	calc2624: LREAL :=  10;
	calc2625: LREAL :=  10;
	calc2626: LREAL :=  10;
	calc2627: LREAL :=  10;
	calc2628: LREAL :=  10;
	calc2629: LREAL :=  10;
	calc2630: LREAL :=  10;
	calc2631: LREAL :=  10;
	calc2632: LREAL :=  10;
	calc2633: LREAL :=  10;
	calc2634: LREAL :=  10;
	calc2635: LREAL :=  10;
	calc2636: LREAL :=  10;
	calc2637: LREAL :=  10;
	calc2638: LREAL :=  10;
	calc2639: LREAL :=  10;
	calc2640: LREAL :=  10;
	calc2641: LREAL :=  10;
	calc2642: LREAL :=  10;
	calc2643: LREAL :=  10;
	calc2644: LREAL :=  10;
	calc2645: LREAL :=  10;
	calc2646: LREAL :=  10;
	calc2647: LREAL :=  10;
	calc2648: LREAL :=  10;
	calc2649: LREAL :=  10;
	calc2650: LREAL :=  10;
	calc2651: LREAL :=  10;
	calc2652: LREAL :=  10;
	calc2653: LREAL :=  10;
	calc2654: LREAL :=  10;
	calc2655: LREAL :=  10;
	calc2656: LREAL :=  10;
	calc2657: LREAL :=  10;
	calc2658: LREAL :=  10;
	calc2659: LREAL :=  10;
	calc2660: LREAL :=  10;
	calc2661: LREAL :=  10;
	calc2662: LREAL :=  10;
	calc2663: LREAL :=  10;
	calc2664: LREAL :=  10;
	calc2665: LREAL :=  10;
	calc2666: LREAL :=  10;
	calc2667: LREAL :=  10;
	calc2668: LREAL :=  10;
	calc2669: LREAL :=  10;
	calc2670: LREAL :=  10;
	calc2671: LREAL :=  10;
	calc2672: LREAL :=  10;
	calc2673: LREAL :=  10;
	calc2674: LREAL :=  10;
	calc2675: LREAL :=  10;
	calc2676: LREAL :=  10;
	calc2677: LREAL :=  10;
	calc2678: LREAL :=  10;
	calc2679: LREAL :=  10;
	calc2680: LREAL :=  10;
	calc2681: LREAL :=  10;
	calc2682: LREAL :=  10;
	calc2683: LREAL :=  10;
	calc2684: LREAL :=  10;
	calc2685: LREAL :=  10;
	calc2686: LREAL :=  10;
	calc2687: LREAL :=  10;
	calc2688: LREAL :=  10;
	calc2689: LREAL :=  10;
	calc2690: LREAL :=  10;
	calc2691: LREAL :=  10;
	calc2692: LREAL :=  10;
	calc2693: LREAL :=  10;
	calc2694: LREAL :=  10;
	calc2695: LREAL :=  10;
	calc2696: LREAL :=  10;
	calc2697: LREAL :=  10;
	calc2698: LREAL :=  10;
	calc2699: LREAL :=  10;
	calc2700: LREAL :=  10;
	calc2701: LREAL :=  10;
	calc2702: LREAL :=  10;
	calc2703: LREAL :=  10;
	calc2704: LREAL :=  10;
	calc2705: LREAL :=  10;
	calc2706: LREAL :=  10;
	calc2707: LREAL :=  10;
	calc2708: LREAL :=  10;
	calc2709: LREAL :=  10;
	calc2710: LREAL :=  10;
	calc2711: LREAL :=  10;
	calc2712: LREAL :=  10;
	calc2713: LREAL :=  10;
	calc2714: LREAL :=  10;
	calc2715: LREAL :=  10;
	calc2716: LREAL :=  10;
	calc2717: LREAL :=  10;
	calc2718: LREAL :=  10;
	calc2719: LREAL :=  10;
	calc2720: LREAL :=  10;
	calc2721: LREAL :=  10;
	calc2722: LREAL :=  10;
	calc2723: LREAL :=  10;
	calc2724: LREAL :=  10;
	calc2725: LREAL :=  10;
	calc2726: LREAL :=  10;
	calc2727: LREAL :=  10;
	calc2728: LREAL :=  10;
	calc2729: LREAL :=  10;
	calc2730: LREAL :=  10;
	calc2731: LREAL :=  10;
	calc2732: LREAL :=  10;
	calc2733: LREAL :=  10;
	calc2734: LREAL :=  10;
	calc2735: LREAL :=  10;
	calc2736: LREAL :=  10;
	calc2737: LREAL :=  10;
	calc2738: LREAL :=  10;
	calc2739: LREAL :=  10;
	calc2740: LREAL :=  10;
	calc2741: LREAL :=  10;
	calc2742: LREAL :=  10;
	calc2743: LREAL :=  10;
	calc2744: LREAL :=  10;
	calc2745: LREAL :=  10;
	calc2746: LREAL :=  10;
	calc2747: LREAL :=  10;
	calc2748: LREAL :=  10;
	calc2749: LREAL :=  10;
	calc2750: LREAL :=  10;
	calc2751: LREAL :=  10;
	calc2752: LREAL :=  10;
	calc2753: LREAL :=  10;
	calc2754: LREAL :=  10;
	calc2755: LREAL :=  10;
	calc2756: LREAL :=  10;
	calc2757: LREAL :=  10;
	calc2758: LREAL :=  10;
	calc2759: LREAL :=  10;
	calc2760: LREAL :=  10;
	calc2761: LREAL :=  10;
	calc2762: LREAL :=  10;
	calc2763: LREAL :=  10;
	calc2764: LREAL :=  10;
	calc2765: LREAL :=  10;
	calc2766: LREAL :=  10;
	calc2767: LREAL :=  10;
	calc2768: LREAL :=  10;
	calc2769: LREAL :=  10;
	calc2770: LREAL :=  10;
	calc2771: LREAL :=  10;
	calc2772: LREAL :=  10;
	calc2773: LREAL :=  10;
	calc2774: LREAL :=  10;
	calc2775: LREAL :=  10;
	calc2776: LREAL :=  10;
	calc2777: LREAL :=  10;
	calc2778: LREAL :=  10;
	calc2779: LREAL :=  10;
	calc2780: LREAL :=  10;
	calc2781: LREAL :=  10;
	calc2782: LREAL :=  10;
	calc2783: LREAL :=  10;
	calc2784: LREAL :=  10;
	calc2785: LREAL :=  10;
	calc2786: LREAL :=  10;
	calc2787: LREAL :=  10;
	calc2788: LREAL :=  10;
	calc2789: LREAL :=  10;
	calc2790: LREAL :=  10;
	calc2791: LREAL :=  10;
	calc2792: LREAL :=  10;
	calc2793: LREAL :=  10;
	calc2794: LREAL :=  10;
	calc2795: LREAL :=  10;
	calc2796: LREAL :=  10;
	calc2797: LREAL :=  10;
	calc2798: LREAL :=  10;
	calc2799: LREAL :=  10;
	calc2800: LREAL :=  10;
	calc2801: LREAL :=  10;
	calc2802: LREAL :=  10;
	calc2803: LREAL :=  10;
	calc2804: LREAL :=  10;
	calc2805: LREAL :=  10;
	calc2806: LREAL :=  10;
	calc2807: LREAL :=  10;
	calc2808: LREAL :=  10;
	calc2809: LREAL :=  10;
	calc2810: LREAL :=  10;
	calc2811: LREAL :=  10;
	calc2812: LREAL :=  10;
	calc2813: LREAL :=  10;
	calc2814: LREAL :=  10;
	calc2815: LREAL :=  10;
	calc2816: LREAL :=  10;
	calc2817: LREAL :=  10;
	calc2818: LREAL :=  10;
	calc2819: LREAL :=  10;
	calc2820: LREAL :=  10;
	calc2821: LREAL :=  10;
	calc2822: LREAL :=  10;
	calc2823: LREAL :=  10;
	calc2824: LREAL :=  10;
	calc2825: LREAL :=  10;
	calc2826: LREAL :=  10;
	calc2827: LREAL :=  10;
	calc2828: LREAL :=  10;
	calc2829: LREAL :=  10;
	calc2830: LREAL :=  10;
	calc2831: LREAL :=  10;
	calc2832: LREAL :=  10;
	calc2833: LREAL :=  10;
	calc2834: LREAL :=  10;
	calc2835: LREAL :=  10;
	calc2836: LREAL :=  10;
	calc2837: LREAL :=  10;
	calc2838: LREAL :=  10;
	calc2839: LREAL :=  10;
	calc2840: LREAL :=  10;
	calc2841: LREAL :=  10;
	calc2842: LREAL :=  10;
	calc2843: LREAL :=  10;
	calc2844: LREAL :=  10;
	calc2845: LREAL :=  10;
	calc2846: LREAL :=  10;
	calc2847: LREAL :=  10;
	calc2848: LREAL :=  10;
	calc2849: LREAL :=  10;
	calc2850: LREAL :=  10;
	calc2851: LREAL :=  10;
	calc2852: LREAL :=  10;
	calc2853: LREAL :=  10;
	calc2854: LREAL :=  10;
	calc2855: LREAL :=  10;
	calc2856: LREAL :=  10;
	calc2857: LREAL :=  10;
	calc2858: LREAL :=  10;
	calc2859: LREAL :=  10;
	calc2860: LREAL :=  10;
	calc2861: LREAL :=  10;
	calc2862: LREAL :=  10;
	calc2863: LREAL :=  10;
	calc2864: LREAL :=  10;
	calc2865: LREAL :=  10;
	calc2866: LREAL :=  10;
	calc2867: LREAL :=  10;
	calc2868: LREAL :=  10;
	calc2869: LREAL :=  10;
	calc2870: LREAL :=  10;
	calc2871: LREAL :=  10;
	calc2872: LREAL :=  10;
	calc2873: LREAL :=  10;
	calc2874: LREAL :=  10;
	calc2875: LREAL :=  10;
	calc2876: LREAL :=  10;
	calc2877: LREAL :=  10;
	calc2878: LREAL :=  10;
	calc2879: LREAL :=  10;
	calc2880: LREAL :=  10;
	calc2881: LREAL :=  10;
	calc2882: LREAL :=  10;
	calc2883: LREAL :=  10;
	calc2884: LREAL :=  10;
	calc2885: LREAL :=  10;
	calc2886: LREAL :=  10;
	calc2887: LREAL :=  10;
	calc2888: LREAL :=  10;
	calc2889: LREAL :=  10;
	calc2890: LREAL :=  10;
	calc2891: LREAL :=  10;
	calc2892: LREAL :=  10;
	calc2893: LREAL :=  10;
	calc2894: LREAL :=  10;
	calc2895: LREAL :=  10;
	calc2896: LREAL :=  10;
	calc2897: LREAL :=  10;
	calc2898: LREAL :=  10;
	calc2899: LREAL :=  10;
	calc2900: LREAL :=  10;
	calc2901: LREAL :=  10;
	calc2902: LREAL :=  10;
	calc2903: LREAL :=  10;
	calc2904: LREAL :=  10;
	calc2905: LREAL :=  10;
	calc2906: LREAL :=  10;
	calc2907: LREAL :=  10;
	calc2908: LREAL :=  10;
	calc2909: LREAL :=  10;
	calc2910: LREAL :=  10;
	calc2911: LREAL :=  10;
	calc2912: LREAL :=  10;
	calc2913: LREAL :=  10;
	calc2914: LREAL :=  10;
	calc2915: LREAL :=  10;
	calc2916: LREAL :=  10;
	calc2917: LREAL :=  10;
	calc2918: LREAL :=  10;
	calc2919: LREAL :=  10;
	calc2920: LREAL :=  10;
	calc2921: LREAL :=  10;
	calc2922: LREAL :=  10;
	calc2923: LREAL :=  10;
	calc2924: LREAL :=  10;
	calc2925: LREAL :=  10;
	calc2926: LREAL :=  10;
	calc2927: LREAL :=  10;
	calc2928: LREAL :=  10;
	calc2929: LREAL :=  10;
	calc2930: LREAL :=  10;
	calc2931: LREAL :=  10;
	calc2932: LREAL :=  10;
	calc2933: LREAL :=  10;
	calc2934: LREAL :=  10;
	calc2935: LREAL :=  10;
	calc2936: LREAL :=  10;
	calc2937: LREAL :=  10;
	calc2938: LREAL :=  10;
	calc2939: LREAL :=  10;
	calc2940: LREAL :=  10;
	calc2941: LREAL :=  10;
	calc2942: LREAL :=  10;
	calc2943: LREAL :=  10;
	calc2944: LREAL :=  10;
	calc2945: LREAL :=  10;
	calc2946: LREAL :=  10;
	calc2947: LREAL :=  10;
	calc2948: LREAL :=  10;
	calc2949: LREAL :=  10;
	calc2950: LREAL :=  10;
	calc2951: LREAL :=  10;
	calc2952: LREAL :=  10;
	calc2953: LREAL :=  10;
	calc2954: LREAL :=  10;
	calc2955: LREAL :=  10;
	calc2956: LREAL :=  10;
	calc2957: LREAL :=  10;
	calc2958: LREAL :=  10;
	calc2959: LREAL :=  10;
	calc2960: LREAL :=  10;
	calc2961: LREAL :=  10;
	calc2962: LREAL :=  10;
	calc2963: LREAL :=  10;
	calc2964: LREAL :=  10;
	calc2965: LREAL :=  10;
	calc2966: LREAL :=  10;
	calc2967: LREAL :=  10;
	calc2968: LREAL :=  10;
	calc2969: LREAL :=  10;
	calc2970: LREAL :=  10;
	calc2971: LREAL :=  10;
	calc2972: LREAL :=  10;
	calc2973: LREAL :=  10;
	calc2974: LREAL :=  10;
	calc2975: LREAL :=  10;
	calc2976: LREAL :=  10;
	calc2977: LREAL :=  10;
	calc2978: LREAL :=  10;
	calc2979: LREAL :=  10;
	calc2980: LREAL :=  10;
	calc2981: LREAL :=  10;
	calc2982: LREAL :=  10;
	calc2983: LREAL :=  10;
	calc2984: LREAL :=  10;
	calc2985: LREAL :=  10;
	calc2986: LREAL :=  10;
	calc2987: LREAL :=  10;
	calc2988: LREAL :=  10;
	calc2989: LREAL :=  10;
	calc2990: LREAL :=  10;
	calc2991: LREAL :=  10;
	calc2992: LREAL :=  10;
	calc2993: LREAL :=  10;
	calc2994: LREAL :=  10;
	calc2995: LREAL :=  10;
	calc2996: LREAL :=  10;
	calc2997: LREAL :=  10;
	calc2998: LREAL :=  10;
	calc2999: LREAL :=  10;
	calc3000: LREAL :=  10;
	calc3001: LREAL :=  10;
	calc3002: LREAL :=  10;
	calc3003: LREAL :=  10;
	calc3004: LREAL :=  10;
	calc3005: LREAL :=  10;
	calc3006: LREAL :=  10;
	calc3007: LREAL :=  10;
	calc3008: LREAL :=  10;
	calc3009: LREAL :=  10;
	calc3010: LREAL :=  10;
	calc3011: LREAL :=  10;
	calc3012: LREAL :=  10;
	calc3013: LREAL :=  10;
	calc3014: LREAL :=  10;
	calc3015: LREAL :=  10;
	calc3016: LREAL :=  10;
	calc3017: LREAL :=  10;
	calc3018: LREAL :=  10;
	calc3019: LREAL :=  10;
	calc3020: LREAL :=  10;
	calc3021: LREAL :=  10;
	calc3022: LREAL :=  10;
	calc3023: LREAL :=  10;
	calc3024: LREAL :=  10;
	calc3025: LREAL :=  10;
	calc3026: LREAL :=  10;
	calc3027: LREAL :=  10;
	calc3028: LREAL :=  10;
	calc3029: LREAL :=  10;
	calc3030: LREAL :=  10;
	calc3031: LREAL :=  10;
	calc3032: LREAL :=  10;
	calc3033: LREAL :=  10;
	calc3034: LREAL :=  10;
	calc3035: LREAL :=  10;
	calc3036: LREAL :=  10;
	calc3037: LREAL :=  10;
	calc3038: LREAL :=  10;
	calc3039: LREAL :=  10;
	calc3040: LREAL :=  10;
	calc3041: LREAL :=  10;
	calc3042: LREAL :=  10;
	calc3043: LREAL :=  10;
	calc3044: LREAL :=  10;
	calc3045: LREAL :=  10;
	calc3046: LREAL :=  10;
	calc3047: LREAL :=  10;
	calc3048: LREAL :=  10;
	calc3049: LREAL :=  10;
	calc3050: LREAL :=  10;
	calc3051: LREAL :=  10;
	calc3052: LREAL :=  10;
	calc3053: LREAL :=  10;
	calc3054: LREAL :=  10;
	calc3055: LREAL :=  10;
	calc3056: LREAL :=  10;
	calc3057: LREAL :=  10;
	calc3058: LREAL :=  10;
	calc3059: LREAL :=  10;
	calc3060: LREAL :=  10;
	calc3061: LREAL :=  10;
	calc3062: LREAL :=  10;
	calc3063: LREAL :=  10;
	calc3064: LREAL :=  10;
	calc3065: LREAL :=  10;
	calc3066: LREAL :=  10;
	calc3067: LREAL :=  10;
	calc3068: LREAL :=  10;
	calc3069: LREAL :=  10;
	calc3070: LREAL :=  10;
	calc3071: LREAL :=  10;
	calc3072: LREAL :=  10;
	calc3073: LREAL :=  10;
	calc3074: LREAL :=  10;
	calc3075: LREAL :=  10;
	calc3076: LREAL :=  10;
	calc3077: LREAL :=  10;
	calc3078: LREAL :=  10;
	calc3079: LREAL :=  10;
	calc3080: LREAL :=  10;
	calc3081: LREAL :=  10;
	calc3082: LREAL :=  10;
	calc3083: LREAL :=  10;
	calc3084: LREAL :=  10;
	calc3085: LREAL :=  10;
	calc3086: LREAL :=  10;
	calc3087: LREAL :=  10;
	calc3088: LREAL :=  10;
	calc3089: LREAL :=  10;
	calc3090: LREAL :=  10;
	calc3091: LREAL :=  10;
	calc3092: LREAL :=  10;
	calc3093: LREAL :=  10;
	calc3094: LREAL :=  10;
	calc3095: LREAL :=  10;
	calc3096: LREAL :=  10;
	calc3097: LREAL :=  10;
	calc3098: LREAL :=  10;
	calc3099: LREAL :=  10;
	calc3100: LREAL :=  10;
	calc3101: LREAL :=  10;
	calc3102: LREAL :=  10;
	calc3103: LREAL :=  10;
	calc3104: LREAL :=  10;
	calc3105: LREAL :=  10;
	calc3106: LREAL :=  10;
	calc3107: LREAL :=  10;
	calc3108: LREAL :=  10;
	calc3109: LREAL :=  10;
	calc3110: LREAL :=  10;
	calc3111: LREAL :=  10;
	calc3112: LREAL :=  10;
	calc3113: LREAL :=  10;
	calc3114: LREAL :=  10;
	calc3115: LREAL :=  10;
	calc3116: LREAL :=  10;
	calc3117: LREAL :=  10;
	calc3118: LREAL :=  10;
	calc3119: LREAL :=  10;
	calc3120: LREAL :=  10;
	calc3121: LREAL :=  10;
	calc3122: LREAL :=  10;
	calc3123: LREAL :=  10;
	calc3124: LREAL :=  10;
	calc3125: LREAL :=  10;
	calc3126: LREAL :=  10;
	calc3127: LREAL :=  10;
	calc3128: LREAL :=  10;
	calc3129: LREAL :=  10;
	calc3130: LREAL :=  10;
	calc3131: LREAL :=  10;
	calc3132: LREAL :=  10;
	calc3133: LREAL :=  10;
	calc3134: LREAL :=  10;
	calc3135: LREAL :=  10;
	calc3136: LREAL :=  10;
	calc3137: LREAL :=  10;
	calc3138: LREAL :=  10;
	calc3139: LREAL :=  10;
	calc3140: LREAL :=  10;
	calc3141: LREAL :=  10;
	calc3142: LREAL :=  10;
	calc3143: LREAL :=  10;
	calc3144: LREAL :=  10;
	calc3145: LREAL :=  10;
	calc3146: LREAL :=  10;
	calc3147: LREAL :=  10;
	calc3148: LREAL :=  10;
	calc3149: LREAL :=  10;
	calc3150: LREAL :=  10;
	calc3151: LREAL :=  10;
	calc3152: LREAL :=  10;
	calc3153: LREAL :=  10;
	calc3154: LREAL :=  10;
	calc3155: LREAL :=  10;
	calc3156: LREAL :=  10;
	calc3157: LREAL :=  10;
	calc3158: LREAL :=  10;
	calc3159: LREAL :=  10;
	calc3160: LREAL :=  10;
	calc3161: LREAL :=  10;
	calc3162: LREAL :=  10;
	calc3163: LREAL :=  10;
	calc3164: LREAL :=  10;
	calc3165: LREAL :=  10;
	calc3166: LREAL :=  10;
	calc3167: LREAL :=  10;
	calc3168: LREAL :=  10;
	calc3169: LREAL :=  10;
	calc3170: LREAL :=  10;
	calc3171: LREAL :=  10;
	calc3172: LREAL :=  10;
	calc3173: LREAL :=  10;
	calc3174: LREAL :=  10;
	calc3175: LREAL :=  10;
	calc3176: LREAL :=  10;
	calc3177: LREAL :=  10;
	calc3178: LREAL :=  10;
	calc3179: LREAL :=  10;
	calc3180: LREAL :=  10;
	calc3181: LREAL :=  10;
	calc3182: LREAL :=  10;
	calc3183: LREAL :=  10;
	calc3184: LREAL :=  10;
	calc3185: LREAL :=  10;
	calc3186: LREAL :=  10;
	calc3187: LREAL :=  10;
	calc3188: LREAL :=  10;
	calc3189: LREAL :=  10;
	calc3190: LREAL :=  10;
	calc3191: LREAL :=  10;
	calc3192: LREAL :=  10;
	calc3193: LREAL :=  10;
	calc3194: LREAL :=  10;
	calc3195: LREAL :=  10;
	calc3196: LREAL :=  10;
	calc3197: LREAL :=  10;
	calc3198: LREAL :=  10;
	calc3199: LREAL :=  10;
	calc3200: LREAL :=  10;
	calc3201: LREAL :=  10;
	calc3202: LREAL :=  10;
	calc3203: LREAL :=  10;
	calc3204: LREAL :=  10;
	calc3205: LREAL :=  10;
	calc3206: LREAL :=  10;
	calc3207: LREAL :=  10;
	calc3208: LREAL :=  10;
	calc3209: LREAL :=  10;
	calc3210: LREAL :=  10;
	calc3211: LREAL :=  10;
	calc3212: LREAL :=  10;
	calc3213: LREAL :=  10;
	calc3214: LREAL :=  10;
	calc3215: LREAL :=  10;
	calc3216: LREAL :=  10;
	calc3217: LREAL :=  10;
	calc3218: LREAL :=  10;
	calc3219: LREAL :=  10;
	calc3220: LREAL :=  10;
	calc3221: LREAL :=  10;
	calc3222: LREAL :=  10;
	calc3223: LREAL :=  10;
	calc3224: LREAL :=  10;
	calc3225: LREAL :=  10;
	calc3226: LREAL :=  10;
	calc3227: LREAL :=  10;
	calc3228: LREAL :=  10;
	calc3229: LREAL :=  10;
	calc3230: LREAL :=  10;
	calc3231: LREAL :=  10;
	calc3232: LREAL :=  10;
	calc3233: LREAL :=  10;
	calc3234: LREAL :=  10;
	calc3235: LREAL :=  10;
	calc3236: LREAL :=  10;
	calc3237: LREAL :=  10;
	calc3238: LREAL :=  10;
	calc3239: LREAL :=  10;
	calc3240: LREAL :=  10;
	calc3241: LREAL :=  10;
	calc3242: LREAL :=  10;
	calc3243: LREAL :=  10;
	calc3244: LREAL :=  10;
	calc3245: LREAL :=  10;
	calc3246: LREAL :=  10;
	calc3247: LREAL :=  10;
	calc3248: LREAL :=  10;
	calc3249: LREAL :=  10;
	calc3250: LREAL :=  10;
	calc3251: LREAL :=  10;
	calc3252: LREAL :=  10;
	calc3253: LREAL :=  10;
	calc3254: LREAL :=  10;
	calc3255: LREAL :=  10;
	calc3256: LREAL :=  10;
	calc3257: LREAL :=  10;
	calc3258: LREAL :=  10;
	calc3259: LREAL :=  10;
	calc3260: LREAL :=  10;
	calc3261: LREAL :=  10;
	calc3262: LREAL :=  10;
	calc3263: LREAL :=  10;
	calc3264: LREAL :=  10;
	calc3265: LREAL :=  10;
	calc3266: LREAL :=  10;
	calc3267: LREAL :=  10;
	calc3268: LREAL :=  10;
	calc3269: LREAL :=  10;
	calc3270: LREAL :=  10;
	calc3271: LREAL :=  10;
	calc3272: LREAL :=  10;
	calc3273: LREAL :=  10;
	calc3274: LREAL :=  10;
	calc3275: LREAL :=  10;
	calc3276: LREAL :=  10;
	calc3277: LREAL :=  10;
	calc3278: LREAL :=  10;
	calc3279: LREAL :=  10;
	calc3280: LREAL :=  10;
	calc3281: LREAL :=  10;
	calc3282: LREAL :=  10;
	calc3283: LREAL :=  10;
	calc3284: LREAL :=  10;
	calc3285: LREAL :=  10;
	calc3286: LREAL :=  10;
	calc3287: LREAL :=  10;
	calc3288: LREAL :=  10;
	calc3289: LREAL :=  10;
	calc3290: LREAL :=  10;
	calc3291: LREAL :=  10;
	calc3292: LREAL :=  10;
	calc3293: LREAL :=  10;
	calc3294: LREAL :=  10;
	calc3295: LREAL :=  10;
	calc3296: LREAL :=  10;
	calc3297: LREAL :=  10;
	calc3298: LREAL :=  10;
	calc3299: LREAL :=  10;
	calc3300: LREAL :=  10;
	calc3301: LREAL :=  10;
	calc3302: LREAL :=  10;
	calc3303: LREAL :=  10;
	calc3304: LREAL :=  10;
	calc3305: LREAL :=  10;
	calc3306: LREAL :=  10;
	calc3307: LREAL :=  10;
	calc3308: LREAL :=  10;
	calc3309: LREAL :=  10;
	calc3310: LREAL :=  10;
	calc3311: LREAL :=  10;
	calc3312: LREAL :=  10;
	calc3313: LREAL :=  10;
	calc3314: LREAL :=  10;
	calc3315: LREAL :=  10;
	calc3316: LREAL :=  10;
	calc3317: LREAL :=  10;
	calc3318: LREAL :=  10;
	calc3319: LREAL :=  10;
	calc3320: LREAL :=  10;
	calc3321: LREAL :=  10;
	calc3322: LREAL :=  10;
	calc3323: LREAL :=  10;
	calc3324: LREAL :=  10;
	calc3325: LREAL :=  10;
	calc3326: LREAL :=  10;
	calc3327: LREAL :=  10;
	calc3328: LREAL :=  10;
	calc3329: LREAL :=  10;
	calc3330: LREAL :=  10;
	calc3331: LREAL :=  10;
	calc3332: LREAL :=  10;
	calc3333: LREAL :=  10;
	calc3334: LREAL :=  10;
	calc3335: LREAL :=  10;
	calc3336: LREAL :=  10;
	calc3337: LREAL :=  10;
	calc3338: LREAL :=  10;
	calc3339: LREAL :=  10;
	calc3340: LREAL :=  10;
	calc3341: LREAL :=  10;
	calc3342: LREAL :=  10;
	calc3343: LREAL :=  10;
	calc3344: LREAL :=  10;
	calc3345: LREAL :=  10;
	calc3346: LREAL :=  10;
	calc3347: LREAL :=  10;
	calc3348: LREAL :=  10;
	calc3349: LREAL :=  10;
	calc3350: LREAL :=  10;
	calc3351: LREAL :=  10;
	calc3352: LREAL :=  10;
	calc3353: LREAL :=  10;
	calc3354: LREAL :=  10;
	calc3355: LREAL :=  10;
	calc3356: LREAL :=  10;
	calc3357: LREAL :=  10;
	calc3358: LREAL :=  10;
	calc3359: LREAL :=  10;
	calc3360: LREAL :=  10;
	calc3361: LREAL :=  10;
	calc3362: LREAL :=  10;
	calc3363: LREAL :=  10;
	calc3364: LREAL :=  10;
	calc3365: LREAL :=  10;
	calc3366: LREAL :=  10;
	calc3367: LREAL :=  10;
	calc3368: LREAL :=  10;
	calc3369: LREAL :=  10;
	calc3370: LREAL :=  10;
	calc3371: LREAL :=  10;
	calc3372: LREAL :=  10;
	calc3373: LREAL :=  10;
	calc3374: LREAL :=  10;
	calc3375: LREAL :=  10;
	calc3376: LREAL :=  10;
	calc3377: LREAL :=  10;
	calc3378: LREAL :=  10;
	calc3379: LREAL :=  10;
	calc3380: LREAL :=  10;
	calc3381: LREAL :=  10;
	calc3382: LREAL :=  10;
	calc3383: LREAL :=  10;
	calc3384: LREAL :=  10;
	calc3385: LREAL :=  10;
	calc3386: LREAL :=  10;
	calc3387: LREAL :=  10;
	calc3388: LREAL :=  10;
	calc3389: LREAL :=  10;
	calc3390: LREAL :=  10;
	calc3391: LREAL :=  10;
	calc3392: LREAL :=  10;
	calc3393: LREAL :=  10;
	calc3394: LREAL :=  10;
	calc3395: LREAL :=  10;
	calc3396: LREAL :=  10;
	calc3397: LREAL :=  10;
	calc3398: LREAL :=  10;
	calc3399: LREAL :=  10;
	calc3400: LREAL :=  10;
	calc3401: LREAL :=  10;
	calc3402: LREAL :=  10;
	calc3403: LREAL :=  10;
	calc3404: LREAL :=  10;
	calc3405: LREAL :=  10;
	calc3406: LREAL :=  10;
	calc3407: LREAL :=  10;
	calc3408: LREAL :=  10;
	calc3409: LREAL :=  10;
	calc3410: LREAL :=  10;
	calc3411: LREAL :=  10;
	calc3412: LREAL :=  10;
	calc3413: LREAL :=  10;
	calc3414: LREAL :=  10;
	calc3415: LREAL :=  10;
	calc3416: LREAL :=  10;
	calc3417: LREAL :=  10;
	calc3418: LREAL :=  10;
	calc3419: LREAL :=  10;
	calc3420: LREAL :=  10;
	calc3421: LREAL :=  10;
	calc3422: LREAL :=  10;
	calc3423: LREAL :=  10;
	calc3424: LREAL :=  10;
	calc3425: LREAL :=  10;
	calc3426: LREAL :=  10;
	calc3427: LREAL :=  10;
	calc3428: LREAL :=  10;
	calc3429: LREAL :=  10;
	calc3430: LREAL :=  10;
	calc3431: LREAL :=  10;
	calc3432: LREAL :=  10;
	calc3433: LREAL :=  10;
	calc3434: LREAL :=  10;
	calc3435: LREAL :=  10;
	calc3436: LREAL :=  10;
	calc3437: LREAL :=  10;
	calc3438: LREAL :=  10;
	calc3439: LREAL :=  10;
	calc3440: LREAL :=  10;
	calc3441: LREAL :=  10;
	calc3442: LREAL :=  10;
	calc3443: LREAL :=  10;
	calc3444: LREAL :=  10;
	calc3445: LREAL :=  10;
	calc3446: LREAL :=  10;
	calc3447: LREAL :=  10;
	calc3448: LREAL :=  10;
	calc3449: LREAL :=  10;
	calc3450: LREAL :=  10;
	calc3451: LREAL :=  10;
	calc3452: LREAL :=  10;
	calc3453: LREAL :=  10;
	calc3454: LREAL :=  10;
	calc3455: LREAL :=  10;
	calc3456: LREAL :=  10;
	calc3457: LREAL :=  10;
	calc3458: LREAL :=  10;
	calc3459: LREAL :=  10;
	calc3460: LREAL :=  10;
	calc3461: LREAL :=  10;
	calc3462: LREAL :=  10;
	calc3463: LREAL :=  10;
	calc3464: LREAL :=  10;
	calc3465: LREAL :=  10;
	calc3466: LREAL :=  10;
	calc3467: LREAL :=  10;
	calc3468: LREAL :=  10;
	calc3469: LREAL :=  10;
	calc3470: LREAL :=  10;
	calc3471: LREAL :=  10;
	calc3472: LREAL :=  10;
	calc3473: LREAL :=  10;
	calc3474: LREAL :=  10;
	calc3475: LREAL :=  10;
	calc3476: LREAL :=  10;
	calc3477: LREAL :=  10;
	calc3478: LREAL :=  10;
	calc3479: LREAL :=  10;
	calc3480: LREAL :=  10;
	calc3481: LREAL :=  10;
	calc3482: LREAL :=  10;
	calc3483: LREAL :=  10;
	calc3484: LREAL :=  10;
	calc3485: LREAL :=  10;
	calc3486: LREAL :=  10;
	calc3487: LREAL :=  10;
	calc3488: LREAL :=  10;
	calc3489: LREAL :=  10;
	calc3490: LREAL :=  10;
	calc3491: LREAL :=  10;
	calc3492: LREAL :=  10;
	calc3493: LREAL :=  10;
	calc3494: LREAL :=  10;
	calc3495: LREAL :=  10;
	calc3496: LREAL :=  10;
	calc3497: LREAL :=  10;
	calc3498: LREAL :=  10;
	calc3499: LREAL :=  10;
	calc3500: LREAL :=  10;
	calc3501: LREAL :=  10;
	calc3502: LREAL :=  10;
	calc3503: LREAL :=  10;
	calc3504: LREAL :=  10;
	calc3505: LREAL :=  10;
	calc3506: LREAL :=  10;
	calc3507: LREAL :=  10;
	calc3508: LREAL :=  10;
	calc3509: LREAL :=  10;
	calc3510: LREAL :=  10;
	calc3511: LREAL :=  10;
	calc3512: LREAL :=  10;
	calc3513: LREAL :=  10;
	calc3514: LREAL :=  10;
	calc3515: LREAL :=  10;
	calc3516: LREAL :=  10;
	calc3517: LREAL :=  10;
	calc3518: LREAL :=  10;
	calc3519: LREAL :=  10;
	calc3520: LREAL :=  10;
	calc3521: LREAL :=  10;
	calc3522: LREAL :=  10;
	calc3523: LREAL :=  10;
	calc3524: LREAL :=  10;
	calc3525: LREAL :=  10;
	calc3526: LREAL :=  10;
	calc3527: LREAL :=  10;
	calc3528: LREAL :=  10;
	calc3529: LREAL :=  10;
	calc3530: LREAL :=  10;
	calc3531: LREAL :=  10;
	calc3532: LREAL :=  10;
	calc3533: LREAL :=  10;
	calc3534: LREAL :=  10;
	calc3535: LREAL :=  10;
	calc3536: LREAL :=  10;
	calc3537: LREAL :=  10;
	calc3538: LREAL :=  10;
	calc3539: LREAL :=  10;
	calc3540: LREAL :=  10;
	calc3541: LREAL :=  10;
	calc3542: LREAL :=  10;
	calc3543: LREAL :=  10;
	calc3544: LREAL :=  10;
	calc3545: LREAL :=  10;
	calc3546: LREAL :=  10;
	calc3547: LREAL :=  10;
	calc3548: LREAL :=  10;
	calc3549: LREAL :=  10;
	calc3550: LREAL :=  10;
	calc3551: LREAL :=  10;
	calc3552: LREAL :=  10;
	calc3553: LREAL :=  10;
	calc3554: LREAL :=  10;
	calc3555: LREAL :=  10;
	calc3556: LREAL :=  10;
	calc3557: LREAL :=  10;
	calc3558: LREAL :=  10;
	calc3559: LREAL :=  10;
	calc3560: LREAL :=  10;
	calc3561: LREAL :=  10;
	calc3562: LREAL :=  10;
	calc3563: LREAL :=  10;
	calc3564: LREAL :=  10;
	calc3565: LREAL :=  10;
	calc3566: LREAL :=  10;
	calc3567: LREAL :=  10;
	calc3568: LREAL :=  10;
	calc3569: LREAL :=  10;
	calc3570: LREAL :=  10;
	calc3571: LREAL :=  10;
	calc3572: LREAL :=  10;
	calc3573: LREAL :=  10;
	calc3574: LREAL :=  10;
	calc3575: LREAL :=  10;
	calc3576: LREAL :=  10;
	calc3577: LREAL :=  10;
	calc3578: LREAL :=  10;
	calc3579: LREAL :=  10;
	calc3580: LREAL :=  10;
	calc3581: LREAL :=  10;
	calc3582: LREAL :=  10;
	calc3583: LREAL :=  10;
	calc3584: LREAL :=  10;
	calc3585: LREAL :=  10;
	calc3586: LREAL :=  10;
	calc3587: LREAL :=  10;
	calc3588: LREAL :=  10;
	calc3589: LREAL :=  10;
	calc3590: LREAL :=  10;
	calc3591: LREAL :=  10;
	calc3592: LREAL :=  10;
	calc3593: LREAL :=  10;
	calc3594: LREAL :=  10;
	calc3595: LREAL :=  10;
	calc3596: LREAL :=  10;
	calc3597: LREAL :=  10;
	calc3598: LREAL :=  10;
	calc3599: LREAL :=  10;
	calc3600: LREAL :=  10;
	calc3601: LREAL :=  10;
	calc3602: LREAL :=  10;
	calc3603: LREAL :=  10;
	calc3604: LREAL :=  10;
	calc3605: LREAL :=  10;
	calc3606: LREAL :=  10;
	calc3607: LREAL :=  10;
	calc3608: LREAL :=  10;
	calc3609: LREAL :=  10;
	calc3610: LREAL :=  10;
	calc3611: LREAL :=  10;
	calc3612: LREAL :=  10;
	calc3613: LREAL :=  10;
	calc3614: LREAL :=  10;
	calc3615: LREAL :=  10;
	calc3616: LREAL :=  10;
	calc3617: LREAL :=  10;
	calc3618: LREAL :=  10;
	calc3619: LREAL :=  10;
	calc3620: LREAL :=  10;
	calc3621: LREAL :=  10;
	calc3622: LREAL :=  10;
	calc3623: LREAL :=  10;
	calc3624: LREAL :=  10;
	calc3625: LREAL :=  10;
	calc3626: LREAL :=  10;
	calc3627: LREAL :=  10;
	calc3628: LREAL :=  10;
	calc3629: LREAL :=  10;
	calc3630: LREAL :=  10;
	calc3631: LREAL :=  10;
	calc3632: LREAL :=  10;
	calc3633: LREAL :=  10;
	calc3634: LREAL :=  10;
	calc3635: LREAL :=  10;
	calc3636: LREAL :=  10;
	calc3637: LREAL :=  10;
	calc3638: LREAL :=  10;
	calc3639: LREAL :=  10;
	calc3640: LREAL :=  10;
	calc3641: LREAL :=  10;
	calc3642: LREAL :=  10;
	calc3643: LREAL :=  10;
	calc3644: LREAL :=  10;
	calc3645: LREAL :=  10;
	calc3646: LREAL :=  10;
	calc3647: LREAL :=  10;
	calc3648: LREAL :=  10;
	calc3649: LREAL :=  10;
	calc3650: LREAL :=  10;
	calc3651: LREAL :=  10;
	calc3652: LREAL :=  10;
	calc3653: LREAL :=  10;
	calc3654: LREAL :=  10;
	calc3655: LREAL :=  10;
	calc3656: LREAL :=  10;
	calc3657: LREAL :=  10;
	calc3658: LREAL :=  10;
	calc3659: LREAL :=  10;
	calc3660: LREAL :=  10;
	calc3661: LREAL :=  10;
	calc3662: LREAL :=  10;
	calc3663: LREAL :=  10;
	calc3664: LREAL :=  10;
	calc3665: LREAL :=  10;
	calc3666: LREAL :=  10;
	calc3667: LREAL :=  10;
	calc3668: LREAL :=  10;
	calc3669: LREAL :=  10;
	calc3670: LREAL :=  10;
	calc3671: LREAL :=  10;
	calc3672: LREAL :=  10;
	calc3673: LREAL :=  10;
	calc3674: LREAL :=  10;
	calc3675: LREAL :=  10;
	calc3676: LREAL :=  10;
	calc3677: LREAL :=  10;
	calc3678: LREAL :=  10;
	calc3679: LREAL :=  10;
	calc3680: LREAL :=  10;
	calc3681: LREAL :=  10;
	calc3682: LREAL :=  10;
	calc3683: LREAL :=  10;
	calc3684: LREAL :=  10;
	calc3685: LREAL :=  10;
	calc3686: LREAL :=  10;
	calc3687: LREAL :=  10;
	calc3688: LREAL :=  10;
	calc3689: LREAL :=  10;
	calc3690: LREAL :=  10;
	calc3691: LREAL :=  10;
	calc3692: LREAL :=  10;
	calc3693: LREAL :=  10;
	calc3694: LREAL :=  10;
	calc3695: LREAL :=  10;
	calc3696: LREAL :=  10;
	calc3697: LREAL :=  10;
	calc3698: LREAL :=  10;
	calc3699: LREAL :=  10;
	calc3700: LREAL :=  10;
	calc3701: LREAL :=  10;
	calc3702: LREAL :=  10;
	calc3703: LREAL :=  10;
	calc3704: LREAL :=  10;
	calc3705: LREAL :=  10;
	calc3706: LREAL :=  10;
	calc3707: LREAL :=  10;
	calc3708: LREAL :=  10;
	calc3709: LREAL :=  10;
	calc3710: LREAL :=  10;
	calc3711: LREAL :=  10;
	calc3712: LREAL :=  10;
	calc3713: LREAL :=  10;
	calc3714: LREAL :=  10;
	calc3715: LREAL :=  10;
	calc3716: LREAL :=  10;
	calc3717: LREAL :=  10;
	calc3718: LREAL :=  10;
	calc3719: LREAL :=  10;
	calc3720: LREAL :=  10;
	calc3721: LREAL :=  10;
	calc3722: LREAL :=  10;
	calc3723: LREAL :=  10;
	calc3724: LREAL :=  10;
	calc3725: LREAL :=  10;
	calc3726: LREAL :=  10;
	calc3727: LREAL :=  10;
	calc3728: LREAL :=  10;
	calc3729: LREAL :=  10;
	calc3730: LREAL :=  10;
	calc3731: LREAL :=  10;
	calc3732: LREAL :=  10;
	calc3733: LREAL :=  10;
	calc3734: LREAL :=  10;
	calc3735: LREAL :=  10;
	calc3736: LREAL :=  10;
	calc3737: LREAL :=  10;
	calc3738: LREAL :=  10;
	calc3739: LREAL :=  10;
	calc3740: LREAL :=  10;
	calc3741: LREAL :=  10;
	calc3742: LREAL :=  10;
	calc3743: LREAL :=  10;
	calc3744: LREAL :=  10;
	calc3745: LREAL :=  10;
	calc3746: LREAL :=  10;
	calc3747: LREAL :=  10;
	calc3748: LREAL :=  10;
	calc3749: LREAL :=  10;
	calc3750: LREAL :=  10;
	calc3751: LREAL :=  10;
	calc3752: LREAL :=  10;
	calc3753: LREAL :=  10;
	calc3754: LREAL :=  10;
	calc3755: LREAL :=  10;
	calc3756: LREAL :=  10;
	calc3757: LREAL :=  10;
	calc3758: LREAL :=  10;
	calc3759: LREAL :=  10;
	calc3760: LREAL :=  10;
	calc3761: LREAL :=  10;
	calc3762: LREAL :=  10;
	calc3763: LREAL :=  10;
	calc3764: LREAL :=  10;
	calc3765: LREAL :=  10;
	calc3766: LREAL :=  10;
	calc3767: LREAL :=  10;
	calc3768: LREAL :=  10;
	calc3769: LREAL :=  10;
	calc3770: LREAL :=  10;
	calc3771: LREAL :=  10;
	calc3772: LREAL :=  10;
	calc3773: LREAL :=  10;
	calc3774: LREAL :=  10;
	calc3775: LREAL :=  10;
	calc3776: LREAL :=  10;
	calc3777: LREAL :=  10;
	calc3778: LREAL :=  10;
	calc3779: LREAL :=  10;
	calc3780: LREAL :=  10;
	calc3781: LREAL :=  10;
	calc3782: LREAL :=  10;
	calc3783: LREAL :=  10;
	calc3784: LREAL :=  10;
	calc3785: LREAL :=  10;
	calc3786: LREAL :=  10;
	calc3787: LREAL :=  10;
	calc3788: LREAL :=  10;
	calc3789: LREAL :=  10;
	calc3790: LREAL :=  10;
	calc3791: LREAL :=  10;
	calc3792: LREAL :=  10;
	calc3793: LREAL :=  10;
	calc3794: LREAL :=  10;
	calc3795: LREAL :=  10;
	calc3796: LREAL :=  10;
	calc3797: LREAL :=  10;
	calc3798: LREAL :=  10;
	calc3799: LREAL :=  10;
	calc3800: LREAL :=  10;
	calc3801: LREAL :=  10;
	calc3802: LREAL :=  10;
	calc3803: LREAL :=  10;
	calc3804: LREAL :=  10;
	calc3805: LREAL :=  10;
	calc3806: LREAL :=  10;
	calc3807: LREAL :=  10;
	calc3808: LREAL :=  10;
	calc3809: LREAL :=  10;
	calc3810: LREAL :=  10;
	calc3811: LREAL :=  10;
	calc3812: LREAL :=  10;
	calc3813: LREAL :=  10;
	calc3814: LREAL :=  10;
	calc3815: LREAL :=  10;
	calc3816: LREAL :=  10;
	calc3817: LREAL :=  10;
	calc3818: LREAL :=  10;
	calc3819: LREAL :=  10;
	calc3820: LREAL :=  10;
	calc3821: LREAL :=  10;
	calc3822: LREAL :=  10;
	calc3823: LREAL :=  10;
	calc3824: LREAL :=  10;
	calc3825: LREAL :=  10;
	calc3826: LREAL :=  10;
	calc3827: LREAL :=  10;
	calc3828: LREAL :=  10;
	calc3829: LREAL :=  10;
	calc3830: LREAL :=  10;
	calc3831: LREAL :=  10;
	calc3832: LREAL :=  10;
	calc3833: LREAL :=  10;
	calc3834: LREAL :=  10;
	calc3835: LREAL :=  10;
	calc3836: LREAL :=  10;
	calc3837: LREAL :=  10;
	calc3838: LREAL :=  10;
	calc3839: LREAL :=  10;
	calc3840: LREAL :=  10;
	calc3841: LREAL :=  10;
	calc3842: LREAL :=  10;
	calc3843: LREAL :=  10;
	calc3844: LREAL :=  10;
	calc3845: LREAL :=  10;
	calc3846: LREAL :=  10;
	calc3847: LREAL :=  10;
	calc3848: LREAL :=  10;
	calc3849: LREAL :=  10;
	calc3850: LREAL :=  10;
	calc3851: LREAL :=  10;
	calc3852: LREAL :=  10;
	calc3853: LREAL :=  10;
	calc3854: LREAL :=  10;
	calc3855: LREAL :=  10;
	calc3856: LREAL :=  10;
	calc3857: LREAL :=  10;
	calc3858: LREAL :=  10;
	calc3859: LREAL :=  10;
	calc3860: LREAL :=  10;
	calc3861: LREAL :=  10;
	calc3862: LREAL :=  10;
	calc3863: LREAL :=  10;
	calc3864: LREAL :=  10;
	calc3865: LREAL :=  10;
	calc3866: LREAL :=  10;
	calc3867: LREAL :=  10;
	calc3868: LREAL :=  10;
	calc3869: LREAL :=  10;
	calc3870: LREAL :=  10;
	calc3871: LREAL :=  10;
	calc3872: LREAL :=  10;
	calc3873: LREAL :=  10;
	calc3874: LREAL :=  10;
	calc3875: LREAL :=  10;
	calc3876: LREAL :=  10;
	calc3877: LREAL :=  10;
	calc3878: LREAL :=  10;
	calc3879: LREAL :=  10;
	calc3880: LREAL :=  10;
	calc3881: LREAL :=  10;
	calc3882: LREAL :=  10;
	calc3883: LREAL :=  10;
	calc3884: LREAL :=  10;
	calc3885: LREAL :=  10;
	calc3886: LREAL :=  10;
	calc3887: LREAL :=  10;
	calc3888: LREAL :=  10;
	calc3889: LREAL :=  10;
	calc3890: LREAL :=  10;
	calc3891: LREAL :=  10;
	calc3892: LREAL :=  10;
	calc3893: LREAL :=  10;
	calc3894: LREAL :=  10;
	calc3895: LREAL :=  10;
	calc3896: LREAL :=  10;
	calc3897: LREAL :=  10;
	calc3898: LREAL :=  10;
	calc3899: LREAL :=  10;
	calc3900: LREAL :=  10;
	calc3901: LREAL :=  10;
	calc3902: LREAL :=  10;
	calc3903: LREAL :=  10;
	calc3904: LREAL :=  10;
	calc3905: LREAL :=  10;
	calc3906: LREAL :=  10;
	calc3907: LREAL :=  10;
	calc3908: LREAL :=  10;
	calc3909: LREAL :=  10;
	calc3910: LREAL :=  10;
	calc3911: LREAL :=  10;
	calc3912: LREAL :=  10;
	calc3913: LREAL :=  10;
	calc3914: LREAL :=  10;
	calc3915: LREAL :=  10;
	calc3916: LREAL :=  10;
	calc3917: LREAL :=  10;
	calc3918: LREAL :=  10;
	calc3919: LREAL :=  10;
	calc3920: LREAL :=  10;
	calc3921: LREAL :=  10;
	calc3922: LREAL :=  10;
	calc3923: LREAL :=  10;
	calc3924: LREAL :=  10;
	calc3925: LREAL :=  10;
	calc3926: LREAL :=  10;
	calc3927: LREAL :=  10;
	calc3928: LREAL :=  10;
	calc3929: LREAL :=  10;
	calc3930: LREAL :=  10;
	calc3931: LREAL :=  10;
	calc3932: LREAL :=  10;
	calc3933: LREAL :=  10;
	calc3934: LREAL :=  10;
	calc3935: LREAL :=  10;
	calc3936: LREAL :=  10;
	calc3937: LREAL :=  10;
	calc3938: LREAL :=  10;
	calc3939: LREAL :=  10;
	calc3940: LREAL :=  10;
	calc3941: LREAL :=  10;
	calc3942: LREAL :=  10;
	calc3943: LREAL :=  10;
	calc3944: LREAL :=  10;
	calc3945: LREAL :=  10;
	calc3946: LREAL :=  10;
	calc3947: LREAL :=  10;
	calc3948: LREAL :=  10;
	calc3949: LREAL :=  10;
	calc3950: LREAL :=  10;
	calc3951: LREAL :=  10;
	calc3952: LREAL :=  10;
	calc3953: LREAL :=  10;
	calc3954: LREAL :=  10;
	calc3955: LREAL :=  10;
	calc3956: LREAL :=  10;
	calc3957: LREAL :=  10;
	calc3958: LREAL :=  10;
	calc3959: LREAL :=  10;
	calc3960: LREAL :=  10;
	calc3961: LREAL :=  10;
	calc3962: LREAL :=  10;
	calc3963: LREAL :=  10;
	calc3964: LREAL :=  10;
	calc3965: LREAL :=  10;
	calc3966: LREAL :=  10;
	calc3967: LREAL :=  10;
	calc3968: LREAL :=  10;
	calc3969: LREAL :=  10;
	calc3970: LREAL :=  10;
	calc3971: LREAL :=  10;
	calc3972: LREAL :=  10;
	calc3973: LREAL :=  10;
	calc3974: LREAL :=  10;
	calc3975: LREAL :=  10;
	calc3976: LREAL :=  10;
	calc3977: LREAL :=  10;
	calc3978: LREAL :=  10;
	calc3979: LREAL :=  10;
	calc3980: LREAL :=  10;
	calc3981: LREAL :=  10;
	calc3982: LREAL :=  10;
	calc3983: LREAL :=  10;
	calc3984: LREAL :=  10;
	calc3985: LREAL :=  10;
	calc3986: LREAL :=  10;
	calc3987: LREAL :=  10;
	calc3988: LREAL :=  10;
	calc3989: LREAL :=  10;
	calc3990: LREAL :=  10;
	calc3991: LREAL :=  10;
	calc3992: LREAL :=  10;
	calc3993: LREAL :=  10;
	calc3994: LREAL :=  10;
	calc3995: LREAL :=  10;
	calc3996: LREAL :=  10;
	calc3997: LREAL :=  10;
	calc3998: LREAL :=  10;
	calc3999: LREAL :=  10;
	calc4000: LREAL :=  10;
	calc4001: LREAL :=  10;
	calc4002: LREAL :=  10;
	calc4003: LREAL :=  10;
	calc4004: LREAL :=  10;
	calc4005: LREAL :=  10;
	calc4006: LREAL :=  10;
	calc4007: LREAL :=  10;
	calc4008: LREAL :=  10;
	calc4009: LREAL :=  10;
	calc4010: LREAL :=  10;
	calc4011: LREAL :=  10;
	calc4012: LREAL :=  10;
	calc4013: LREAL :=  10;
	calc4014: LREAL :=  10;
	calc4015: LREAL :=  10;
	calc4016: LREAL :=  10;
	calc4017: LREAL :=  10;
	calc4018: LREAL :=  10;
	calc4019: LREAL :=  10;
	calc4020: LREAL :=  10;
	calc4021: LREAL :=  10;
	calc4022: LREAL :=  10;
	calc4023: LREAL :=  10;
	calc4024: LREAL :=  10;
	calc4025: LREAL :=  10;
	calc4026: LREAL :=  10;
	calc4027: LREAL :=  10;
	calc4028: LREAL :=  10;
	calc4029: LREAL :=  10;
	calc4030: LREAL :=  10;
	calc4031: LREAL :=  10;
	calc4032: LREAL :=  10;
	calc4033: LREAL :=  10;
	calc4034: LREAL :=  10;
	calc4035: LREAL :=  10;
	calc4036: LREAL :=  10;
	calc4037: LREAL :=  10;
	calc4038: LREAL :=  10;
	calc4039: LREAL :=  10;
	calc4040: LREAL :=  10;
	calc4041: LREAL :=  10;
